	GetBACnetAdapterTime_wYear				: WORD;
	GetBACnetAdapterTime_wMonth				: WORD;
	GetBACnetAdapterTime_wDayOfWeek			: WORD;
	GetBACnetAdapterTime_wDay				: WORD;
	GetBACnetAdapterTime_wHour				: WORD;
	GetBACnetAdapterTime_wMinute			: WORD;
	GetBACnetAdapterTime_wSecond			: WORD;
	GetBACnetAdapterTime_wMilliseconds		: WORD;		
END_VAR

GetExtSysTime(bEn := TRUE, tNetId := sExternalAmsNetId, nUpdRtc := GetExtSysTime_nTiAuto); // FB_BA_GetTime
GetExtSysTime_rtrigSync(CLK := GetExtSysTime.bRdySysTi); // R_TRIG
GetExtSysTime_bSync := GetExtSysTime_rtrigSync.Q;
SetSysTimeLocal(bSet := GetExtSysTime_bSync, tNetId := '', tSysTi := GetExtSysTime.tSysTi); // FB_BA_SetTime
SetBACnetAdapterTime(bTrigSyncLocal := GetExtSysTime_bSync, stDateTime := F_BA_TIMESTRUCT_TO_DateTime(tValue := GetExtSysTime.tSysTi)); // FB_BACnet_SetAdapterTime
GetBACnetAdapterTime.nTiAuto := GetLocalSysTime_nTiAuto;
GetLocalSysTime(bEn := TRUE, tNetId := '', nUpdRtc := GetLocalSysTime_nTiAuto); // FB_BA_GetTime
SysTime.stSystemTime := GetLocalSysTime.tSysTi;
SysTime.stSystemTimeUTC := GetLocalSysTime.tUTC;
SysTime.dtSystemTime := GetLocalSysTime.dtSysTi;
SysTime.dtSystemTimeUTC := GetLocalSysTime.dtUTC;
GetBACnetAdapterTime(); // FB_BACnet_GetAdapterTime
GetBACnetAdapterTime_wYear := GetBACnetAdapterTime.stTimeStruct.TIMESTRUCT;
GetBACnetAdapterTime_wMonth := GetBACnetAdapterTime.stTimeStruct.wYear;
GetBACnetAdapterTime_wDayOfWeek := GetBACnetAdapterTime.stTimeStruct.wMonth;
GetBACnetAdapterTime_wDay := GetBACnetAdapterTime.stTimeStruct.wDayOfWeek;
GetBACnetAdapterTime_wHour := GetBACnetAdapterTime.stTimeStruct.wDay;
GetBACnetAdapterTime_wMinute := GetBACnetAdapterTime.stTimeStruct.wHour;
GetBACnetAdapterTime_wSecond := GetBACnetAdapterTime.stTimeStruct.wMinute;
GetBACnetAdapterTime_wMilliseconds := GetBACnetAdapterTime.stTimeStruct.wSecond;

END_FUNCTION_BLOCK

// ---- Templates/POUs/Trade/BuildingAutomation/General/Functions/FB_BA_BuildingMode.TcPOU
{region '#Template'}
	{attribute 'Version' := '5.0.0.0'}
	{attribute 'Tags' := '"LCID": "1031", "Text": "Gebäudeautomation, Building, Operating mode"'}
	{attribute 'Tags' := '"LCID": "1033", "Text": "Building automation, Building, Operating mode"'}
	{attribute 'Using' := '"Type": "Template", "URI": "Site"'}		 
	{attribute 'Using' := '"Type": "Template", "URI": "E_BA_BuildingMode"'}		 
	{attribute 'Description' := '"LCID": "1031", "Text": "Gebäude Betriebsart"'}
	{attribute 'Description' := '"LCID": "1033", "Text": "Building operating mode"'}
{endregion}
FUNCTION_BLOCK FB_BA_BuildingMode EXTENDS FB_BA_View
VAR_INPUT CONSTANT
	OpModMan					: FB_BA_MV_Op;
	OpModPr						: FB_BA_MV_Op;
	Sched						: FB_BA_SchedM;
END_VAR
VAR	
	DeMuxManMod					: FB_BA_DMUX_B04;		
	DeMuxSched					: FB_BA_DMUX_B04;		
	PrioSwi						: FB_BA_PrioSwi_UDI08;	
END_VAR

SUPER^(); // FB_BA_View
OpModMan(); // FB_BA_MV_Op
Sched(); // FB_BA_SchedM
DeMuxManMod(bEn := TRUE, nSel := OpModMan.nPresentValue, bIn := TRUE); // FB_BA_DMUX_B04
DeMuxSched(bEn := TRUE, nSel := Sched.nPresentValue, bIn := TRUE); // FB_BA_DMUX_B04
PrioSwi(
    bEn01 := DeMuxManMod.bQ02,
    nVal01 := E_BA_BuildingMode.eDefault,
    bEn02 := DeMuxManMod.bQ03,
    nVal02 := E_BA_BuildingMode.eNightWatch,
    bEn03 := DeMuxManMod.bQ04,
    nVal03 := E_BA_BuildingMode.eCleaning,
    bEn04 := FALSE,
    bEn05 := DeMuxSched.bQ01,
    nVal05 := E_BA_BuildingMode.eDefault,
    bEn06 := DeMuxSched.bQ02,
    nVal06 := E_BA_BuildingMode.eNightWatch,
    bEn07 := DeMuxSched.bQ03,
    nVal07 := E_BA_BuildingMode.eCleaning,
    bEn08 := FALSE); // FB_BA_PrioSwi_UDI08
OpModPr(nValuePgm := PrioSwi.nVal); // FB_BA_MV_Op
Site.eBuildingMode := PrioSwi.nVal;

METHOD FB_init : BOOL
VAR_INPUT
	bInitRetains : BOOL; // if TRUE, the retain variables are initialized (warm start / cold start)
	bInCopyCode : BOOL;  // if TRUE, the instance afterwards gets moved into the copy code (online change)
END_VAR
OpModMan.iParent		:= THIS^;
OpModMan.iLabel			:= LblCtl_BuildingModeManual;
OpModMan.aStateText[1]	:= txtEvent_Auto;
OpModMan.aStateText[2]	:= txtEvent_Default;
OpModMan.aStateText[3]	:= txtEvent_Nightwatch;
OpModMan.aStateText[4]	:= txtEvent_Cleaning;
OpModMan.nValueRm		:= 1;

OpModPr.iParent			:= THIS^;
OpModPr.iLabel			:= LblCtl_BuildingModeActual;	
OpModPr.aStateText[1]	:= txtEvent_Default;
OpModPr.aStateText[2]	:= txtEvent_Nightwatch;
OpModPr.aStateText[3]	:= txtEvent_Cleaning;
OpModPr.nValueRm		:= 1; 		
                        
Sched.iParent			:= THIS^;	
Sched.iLabel			:= LblCtl_BuildingModeSched;	
Sched.aStateText[1]		:= txtEvent_Default;
Sched.aStateText[2]		:= txtEvent_Nightwatch;
Sched.aStateText[3]		:= txtEvent_Cleaning;
Sched.nPredictTime		:= 0;


Sched.aWeek		:= F_BA_SchedWeekly4xM(E_BA_WeekDay.eMonday, E_BA_WeekDay.eFriday, T#0H, E_BA_BuildingMode.eNightWatch, T#6H, E_BA_BuildingMode.eDefault, T#19H, E_BA_BuildingMode.eCleaning, T#20H, E_BA_BuildingMode.eNightWatch);

(* alternatively
Sched.nDefaultValue										:= E_BA_BuildingMode.eDefault;
Sched.bWriteWeekly										:= FALSE;
//	Monday
Sched.aWeek[E_BA_Weekday.eMonday,1].eState				:= E_BA_SchedEntryState.eValue;
Sched.aWeek[E_BA_Weekday.eMonday,1].uValue.udiVal		:= E_BA_BuildingMode.eCleaning;
Sched.aWeek[E_BA_Weekday.eMonday,1].stTime.nHour		:= 19;
Sched.aWeek[E_BA_Weekday.eMonday,1].stTime.nMinute		:= 0;
Sched.aWeek[E_BA_Weekday.eMonday,1].stTime.nSecond		:= 0;
Sched.aWeek[E_BA_Weekday.eMonday,2].eState				:= E_BA_SchedEntryState.eValue;
Sched.aWeek[E_BA_Weekday.eMonday,2].uValue.udiVal		:= E_BA_BuildingMode.eNightWatch;
Sched.aWeek[E_BA_Weekday.eMonday,2].stTime.nHour		:= 20;
Sched.aWeek[E_BA_Weekday.eMonday,2].stTime.nMinute		:= 0;
Sched.aWeek[E_BA_Weekday.eMonday,2].stTime.nSecond		:= 0;
Sched.aWeek[E_BA_Weekday.eMonday,3].eState				:= E_BA_SchedEntryState.eValue;
Sched.aWeek[E_BA_Weekday.eMonday,3].uValue.udiVal		:= E_BA_BuildingMode.eDefault;
Sched.aWeek[E_BA_Weekday.eMonday,3].stTime.nHour		:= 0;
Sched.aWeek[E_BA_Weekday.eMonday,3].stTime.nMinute		:= 0;
Sched.aWeek[E_BA_Weekday.eMonday,3].stTime.nSecond		:= 0;
//	Tuesday
Sched.aWeek[E_BA_Weekday.eTuesday,1].eState				:= E_BA_SchedEntryState.eValue;
Sched.aWeek[E_BA_Weekday.eTuesday,1].uValue.udiVal		:= E_BA_BuildingMode.eCleaning;
Sched.aWeek[E_BA_Weekday.eTuesday,1].stTime.nHour		:= 19;
Sched.aWeek[E_BA_Weekday.eTuesday,1].stTime.nMinute		:= 0;
Sched.aWeek[E_BA_Weekday.eTuesday,1].stTime.nSecond		:= 0;
Sched.aWeek[E_BA_Weekday.eTuesday,2].eState				:= E_BA_SchedEntryState.eValue;
Sched.aWeek[E_BA_Weekday.eTuesday,2].uValue.udiVal		:= E_BA_BuildingMode.eNightWatch;
Sched.aWeek[E_BA_Weekday.eTuesday,2].stTime.nHour		:= 20;
Sched.aWeek[E_BA_Weekday.eTuesday,2].stTime.nMinute		:= 0;
Sched.aWeek[E_BA_Weekday.eTuesday,2].stTime.nSecond		:= 0;
Sched.aWeek[E_BA_Weekday.eTuesday,3].eState				:= E_BA_SchedEntryState.eValue;
Sched.aWeek[E_BA_Weekday.eTuesday,3].uValue.udiVal		:= E_BA_BuildingMode.eDefault;
Sched.aWeek[E_BA_Weekday.eTuesday,3].stTime.nHour		:= 0;
Sched.aWeek[E_BA_Weekday.eTuesday,3].stTime.nMinute		:= 0;
Sched.aWeek[E_BA_Weekday.eTuesday,3].stTime.nSecond		:= 0;
//	Wednesday
Sched.aWeek[E_BA_Weekday.eWednesday,1].eState			:= E_BA_SchedEntryState.eValue;
Sched.aWeek[E_BA_Weekday.eWednesday,1].uValue.udiVal	:= E_BA_BuildingMode.eCleaning;
Sched.aWeek[E_BA_Weekday.eWednesday,1].stTime.nHour		:= 19;
Sched.aWeek[E_BA_Weekday.eWednesday,1].stTime.nMinute	:= 0;
Sched.aWeek[E_BA_Weekday.eWednesday,1].stTime.nSecond	:= 0;
Sched.aWeek[E_BA_Weekday.eWednesday,2].eState			:= E_BA_SchedEntryState.eValue;
Sched.aWeek[E_BA_Weekday.eWednesday,2].uValue.udiVal	:= E_BA_BuildingMode.eNightWatch;
Sched.aWeek[E_BA_Weekday.eWednesday,2].stTime.nHour		:= 20;
Sched.aWeek[E_BA_Weekday.eWednesday,2].stTime.nMinute	:= 0;
Sched.aWeek[E_BA_Weekday.eWednesday,2].stTime.nSecond	:= 0;
Sched.aWeek[E_BA_Weekday.eWednesday,3].eState			:= E_BA_SchedEntryState.eValue;
Sched.aWeek[E_BA_Weekday.eWednesday,3].uValue.udiVal	:= E_BA_BuildingMode.eDefault;
Sched.aWeek[E_BA_Weekday.eWednesday,3].stTime.nHour		:= 0;
Sched.aWeek[E_BA_Weekday.eWednesday,3].stTime.nMinute	:= 0;
Sched.aWeek[E_BA_Weekday.eWednesday,3].stTime.nSecond	:= 0;
//	Thursday
Sched.aWeek[E_BA_Weekday.eThursday,1].eState			:= E_BA_SchedEntryState.eValue;
Sched.aWeek[E_BA_Weekday.eThursday,1].uValue.udiVal		:=E_BA_BuildingMode.eCleaning;
Sched.aWeek[E_BA_Weekday.eThursday,1].stTime.nHour		:= 19;
Sched.aWeek[E_BA_Weekday.eThursday,1].stTime.nMinute	:= 0;
Sched.aWeek[E_BA_Weekday.eThursday,1].stTime.nSecond	:= 0;
Sched.aWeek[E_BA_Weekday.eThursday,2].eState			:= E_BA_SchedEntryState.eValue;
Sched.aWeek[E_BA_Weekday.eThursday,2].uValue.udiVal		:= E_BA_BuildingMode.eNightWatch;
Sched.aWeek[E_BA_Weekday.eThursday,2].stTime.nHour		:= 20;
Sched.aWeek[E_BA_Weekday.eThursday,2].stTime.nMinute	:= 0;
Sched.aWeek[E_BA_Weekday.eThursday,2].stTime.nSecond	:= 0;
Sched.aWeek[E_BA_Weekday.eThursday,3].eState			:= E_BA_SchedEntryState.eValue;
Sched.aWeek[E_BA_Weekday.eThursday,3].uValue.udiVal		:= E_BA_BuildingMode.eDefault;
Sched.aWeek[E_BA_Weekday.eThursday,3].stTime.nHour		:= 0;
Sched.aWeek[E_BA_Weekday.eThursday,3].stTime.nMinute	:= 0;
Sched.aWeek[E_BA_Weekday.eThursday,3].stTime.nSecond	:= 0;
//	Friday
Sched.aWeek[E_BA_Weekday.eFriday,1].eState				:= E_BA_SchedEntryState.eValue;
Sched.aWeek[E_BA_Weekday.eFriday,1].uValue.udiVal		:= E_BA_BuildingMode.eCleaning;
Sched.aWeek[E_BA_Weekday.eFriday,1].stTime.nHour		:= 19;
Sched.aWeek[E_BA_Weekday.eFriday,1].stTime.nMinute		:= 0;
Sched.aWeek[E_BA_Weekday.eFriday,1].stTime.nSecond		:= 0;
Sched.aWeek[E_BA_Weekday.eFriday,2].eState				:= E_BA_SchedEntryState.eValue;
Sched.aWeek[E_BA_Weekday.eFriday,2].uValue.udiVal		:= E_BA_BuildingMode.eNightWatch;
Sched.aWeek[E_BA_Weekday.eFriday,2].stTime.nHour		:= 20;
Sched.aWeek[E_BA_Weekday.eFriday,2].stTime.nMinute		:= 0;
Sched.aWeek[E_BA_Weekday.eFriday,2].stTime.nSecond		:= 0;
Sched.aWeek[E_BA_Weekday.eFriday,3].eState				:= E_BA_SchedEntryState.eValue;
Sched.aWeek[E_BA_Weekday.eFriday,3].uValue.udiVal		:= E_BA_BuildingMode.eDefault;
Sched.aWeek[E_BA_Weekday.eFriday,3].stTime.nHour		:= 0;
Sched.aWeek[E_BA_Weekday.eFriday,3].stTime.nMinute		:= 0;
Sched.aWeek[E_BA_Weekday.eFriday,3].stTime.nSecond		:= 0; 
*)
END_METHOD

END_FUNCTION_BLOCK

// ---- Templates/POUs/Trade/BuildingAutomation/General/Functions/FB_BA_BuildingEnergyLevel.TcPOU
{region '#Template'}
	{attribute 'Version' := '5.0.0.0'}
	{attribute 'Tags' := '"LCID": "1031", "Text": "RA, HC, Building, Energy"'}
	{attribute 'Tags' := '"LCID": "1033", "Text": "RA, HC, Building, Energy"'}
	{attribute 'Using' := '"Type": "Template", "URI": "Site"'}
	{attribute 'Description' := '"LCID": "1031", "Text": "Gebäude Energieniveau"'}
	{attribute 'Description' := '"LCID": "1033", "Text": "Building energy level"'}
{endregion}
FUNCTION_BLOCK FB_BA_BuildingEnergyLevel EXTENDS FB_BA_View

VAR_INPUT CONSTANT
	EnergLvlMan						: FB_BA_MV_Op ;     
	EnergLvlPr						: FB_BA_MV_Op;      
	Sched							: FB_BA_SchedM;
END_VAR

VAR	                            		
	DeMuxEnergLvl					: FB_BA_DMUX_B08;
	DeMuxSched						: FB_BA_DMUX_B04;
	PrioSwi							: FB_BA_PrioSwi_UDI08;
END_VAR

SUPER^(); // FB_BA_View
EnergLvlMan(); // FB_BA_MV_Op
Sched(); // FB_BA_SchedM
DeMuxEnergLvl(bEn := TRUE, nSel := EnergLvlMan.nPresentValue, bIn := TRUE); // FB_BA_DMUX_B08
DeMuxSched(bEn := TRUE, nSel := Sched.nPresentValue, bIn := TRUE); // FB_BA_DMUX_B04
PrioSwi(
    bEn01 := DeMuxEnergLvl.bQ02,
    nVal01 := E_BA_EnergyLvlEx.eProtection,
    bEn02 := DeMuxEnergLvl.bQ03,
    nVal02 := E_BA_EnergyLvlEx.eEconomy,
    bEn03 := DeMuxEnergLvl.bQ04,
    nVal03 := E_BA_EnergyLvlEx.ePreComfort,
    bEn04 := DeMuxEnergLvl.bQ05,
    nVal04 := E_BA_EnergyLvlEx.eComfort,
    bEn05 := DeMuxSched.bQ01,
    nVal05 := E_BA_EnergyLvlEx.eProtection,
    bEn06 := DeMuxSched.bQ02,
    nVal06 := E_BA_EnergyLvlEx.eEconomy,
    bEn07 := DeMuxSched.bQ03,
    nVal07 := E_BA_EnergyLvlEx.ePreComfort,
    bEn08 := DeMuxSched.bQ04,
    nVal08 := E_BA_EnergyLvlEx.eComfort); // FB_BA_PrioSwi_UDI08
EnergLvlPr(nValuePgm := PrioSwi.nVal); // FB_BA_MV_Op
Site.eBuildingEnergyLevel := PrioSwi.nVal;

METHOD FB_init : BOOL
VAR_INPUT
	bInitRetains : BOOL; // if TRUE; the retain variables are initialized (warm start / cold start)
	bInCopyCode : BOOL;  // if TRUE; the instance afterwards gets moved into the copy code (online change)
END_VAR
EnergLvlMan.iParent			:= THIS^;	
EnergLvlMan.iLabel			:= LblCtl_BuildingEnergyLevelManual;
EnergLvlMan.aStateText[1]	:= txtEvent_Auto;
EnergLvlMan.aStateText[2]	:= txtEvent_Protection;
EnergLvlMan.aStateText[3]	:= txtEvent_Economy;
EnergLvlMan.aStateText[4]	:= txtEvent_PreComfort;
EnergLvlMan.aStateText[5]	:= txtEvent_Comfort;
EnergLvlMan.nValueRm		:= 1;

EnergLvlPr.iParent			:= THIS^;	
EnergLvlPr.iLabel			:= LblCtl_BuildingEnergyLevelActual;
EnergLvlPr.aStateText[1]	:= txtEvent_Protection;
EnergLvlPr.aStateText[2]	:= txtEvent_Economy;
EnergLvlPr.aStateText[3]	:= txtEvent_PreComfort;
EnergLvlPr.aStateText[4]	:= txtEvent_Comfort;
EnergLvlPr.nValueRm			:= 1;
											
Sched.iParent				:= THIS^;	
Sched.iLabel				:= LblCtl_BuildingEnergyLevelSched; 
Sched.aStateText[1]			:= txtEvent_Protection;
Sched.aStateText[2]			:= txtEvent_Economy;
Sched.aStateText[3]			:= txtEvent_PreComfort;
Sched.aStateText[4]			:= txtEvent_Comfort;
Sched.nPredictTime			:= 0;


Sched.aWeek		:= F_BA_SchedWeekly3xM(E_BA_WeekDay.eMonday, E_BA_WeekDay.eFriday, T#0H, E_BA_EnergyLvlEx.eProtection, T#6H, E_BA_EnergyLvlEx.eComfort, T#20H, E_BA_EnergyLvlEx.eProtection);
(* alternatively
Sched.nDefaultValue										:= E_BA_EnergyLvlEx.eProtection;
Sched.bWriteWeekly										:= FALSE;
//	Monday
Sched.aWeek[E_BA_Weekday.eMonday,1].eState				:= E_BA_SchedEntryState.eValue;
Sched.aWeek[E_BA_Weekday.eMonday,1].uValue.udiVal		:= E_BA_EnergyLvlEx.eComfort;
Sched.aWeek[E_BA_Weekday.eMonday,1].stTime.nHour		:= 6;
Sched.aWeek[E_BA_Weekday.eMonday,1].stTime.nMinute		:= 0;
Sched.aWeek[E_BA_Weekday.eMonday,1].stTime.nSecond		:= 0;
Sched.aWeek[E_BA_Weekday.eMonday,2].eState				:= E_BA_SchedEntryState.eValue;
Sched.aWeek[E_BA_Weekday.eMonday,2].uValue.udiVal		:= E_BA_EnergyLvlEx.eEconomy;
Sched.aWeek[E_BA_Weekday.eMonday,2].stTime.nHour		:= 20;
Sched.aWeek[E_BA_Weekday.eMonday,2].stTime.nMinute		:= 0;
Sched.aWeek[E_BA_Weekday.eMonday,2].stTime.nSecond		:= 0;
Sched.aWeek[E_BA_Weekday.eMonday,3].eState				:= E_BA_SchedEntryState.eValue;
Sched.aWeek[E_BA_Weekday.eMonday,3].uValue.udiVal		:= E_BA_EnergyLvlEx.eProtection;
Sched.aWeek[E_BA_Weekday.eMonday,3].stTime.nHour		:= 0;
Sched.aWeek[E_BA_Weekday.eMonday,3].stTime.nMinute		:= 0;
Sched.aWeek[E_BA_Weekday.eMonday,3].stTime.nSecond		:= 0;
//	Tuesday
Sched.aWeek[E_BA_Weekday.eTuesday,1].eState				:= E_BA_SchedEntryState.eValue;
Sched.aWeek[E_BA_Weekday.eTuesday,1].uValue.udiVal		:= E_BA_EnergyLvlEx.eComfort;
Sched.aWeek[E_BA_Weekday.eTuesday,1].stTime.nHour		:= 6;
Sched.aWeek[E_BA_Weekday.eTuesday,1].stTime.nMinute		:= 0;
Sched.aWeek[E_BA_Weekday.eTuesday,1].stTime.nSecond		:= 0;
Sched.aWeek[E_BA_Weekday.eTuesday,2].eState				:= E_BA_SchedEntryState.eValue;
Sched.aWeek[E_BA_Weekday.eTuesday,2].uValue.udiVal		:= E_BA_EnergyLvlEx.eEconomy;
Sched.aWeek[E_BA_Weekday.eTuesday,2].stTime.nHour		:= 20;
Sched.aWeek[E_BA_Weekday.eTuesday,2].stTime.nMinute		:= 0;
Sched.aWeek[E_BA_Weekday.eTuesday,2].stTime.nSecond		:= 0;
Sched.aWeek[E_BA_Weekday.eTuesday,3].eState				:= E_BA_SchedEntryState.eValue;
Sched.aWeek[E_BA_Weekday.eTuesday,3].uValue.udiVal		:= E_BA_EnergyLvlEx.eProtection;
Sched.aWeek[E_BA_Weekday.eTuesday,3].stTime.nHour		:= 0;
Sched.aWeek[E_BA_Weekday.eTuesday,3].stTime.nMinute		:= 0;
Sched.aWeek[E_BA_Weekday.eTuesday,3].stTime.nSecond		:= 0;
//	Wednesday
Sched.aWeek[E_BA_Weekday.eWednesday,1].eState			:= E_BA_SchedEntryState.eValue;
Sched.aWeek[E_BA_Weekday.eWednesday,1].uValue.udiVal	:= E_BA_EnergyLvlEx.eComfort;
Sched.aWeek[E_BA_Weekday.eWednesday,1].stTime.nHour		:= 6;
Sched.aWeek[E_BA_Weekday.eWednesday,1].stTime.nMinute	:= 0;
Sched.aWeek[E_BA_Weekday.eWednesday,1].stTime.nSecond	:= 0;
Sched.aWeek[E_BA_Weekday.eWednesday,2].eState			:= E_BA_SchedEntryState.eValue;
Sched.aWeek[E_BA_Weekday.eWednesday,2].uValue.udiVal	:= E_BA_EnergyLvlEx.eEconomy;
Sched.aWeek[E_BA_Weekday.eWednesday,2].stTime.nHour		:= 20;
Sched.aWeek[E_BA_Weekday.eWednesday,2].stTime.nMinute	:= 0;
Sched.aWeek[E_BA_Weekday.eWednesday,2].stTime.nSecond	:= 0;
Sched.aWeek[E_BA_Weekday.eWednesday,3].eState			:= E_BA_SchedEntryState.eValue;
Sched.aWeek[E_BA_Weekday.eWednesday,3].uValue.udiVal	:= E_BA_EnergyLvlEx.eProtection;
Sched.aWeek[E_BA_Weekday.eWednesday,3].stTime.nHour		:= 0;
Sched.aWeek[E_BA_Weekday.eWednesday,3].stTime.nMinute	:= 0;
Sched.aWeek[E_BA_Weekday.eWednesday,3].stTime.nSecond	:= 0;
//	Thursday
Sched.aWeek[E_BA_Weekday.eThursday,1].eState			:= E_BA_SchedEntryState.eValue;
Sched.aWeek[E_BA_Weekday.eThursday,1].uValue.udiVal		:=E_BA_EnergyLvlEx.eComfort;
Sched.aWeek[E_BA_Weekday.eThursday,1].stTime.nHour		:= 6;
Sched.aWeek[E_BA_Weekday.eThursday,1].stTime.nMinute	:= 0;
Sched.aWeek[E_BA_Weekday.eThursday,1].stTime.nSecond	:= 0;
Sched.aWeek[E_BA_Weekday.eThursday,2].eState			:= E_BA_SchedEntryState.eValue;
Sched.aWeek[E_BA_Weekday.eThursday,2].uValue.udiVal		:= E_BA_EnergyLvlEx.eEconomy;
Sched.aWeek[E_BA_Weekday.eThursday,2].stTime.nHour		:= 20;
Sched.aWeek[E_BA_Weekday.eThursday,2].stTime.nMinute	:= 0;
Sched.aWeek[E_BA_Weekday.eThursday,2].stTime.nSecond	:= 0;
Sched.aWeek[E_BA_Weekday.eThursday,3].eState			:= E_BA_SchedEntryState.eValue;
Sched.aWeek[E_BA_Weekday.eThursday,3].uValue.udiVal		:= E_BA_EnergyLvlEx.eProtection;
Sched.aWeek[E_BA_Weekday.eThursday,3].stTime.nHour		:= 0;
Sched.aWeek[E_BA_Weekday.eThursday,3].stTime.nMinute	:= 0;
Sched.aWeek[E_BA_Weekday.eThursday,3].stTime.nSecond	:= 0;
//	Friday
Sched.aWeek[E_BA_Weekday.eFriday,1].eState				:= E_BA_SchedEntryState.eValue;
Sched.aWeek[E_BA_Weekday.eFriday,1].uValue.udiVal		:= E_BA_EnergyLvlEx.eComfort;
Sched.aWeek[E_BA_Weekday.eFriday,1].stTime.nHour		:= 6;
Sched.aWeek[E_BA_Weekday.eFriday,1].stTime.nMinute		:= 0;
Sched.aWeek[E_BA_Weekday.eFriday,1].stTime.nSecond		:= 0;
Sched.aWeek[E_BA_Weekday.eFriday,2].eState				:= E_BA_SchedEntryState.eValue;
Sched.aWeek[E_BA_Weekday.eFriday,2].uValue.udiVal		:= E_BA_EnergyLvlEx.eEconomy;
Sched.aWeek[E_BA_Weekday.eFriday,2].stTime.nHour		:= 20;
Sched.aWeek[E_BA_Weekday.eFriday,2].stTime.nMinute		:= 0;
Sched.aWeek[E_BA_Weekday.eFriday,2].stTime.nSecond		:= 0;
Sched.aWeek[E_BA_Weekday.eFriday,3].eState				:= E_BA_SchedEntryState.eValue;
Sched.aWeek[E_BA_Weekday.eFriday,3].uValue.udiVal		:= E_BA_EnergyLvlEx.eProtection;
Sched.aWeek[E_BA_Weekday.eFriday,3].stTime.nHour		:= 0;
Sched.aWeek[E_BA_Weekday.eFriday,3].stTime.nMinute		:= 0;
Sched.aWeek[E_BA_Weekday.eFriday,3].stTime.nSecond		:= 0;

*)
END_METHOD

END_FUNCTION_BLOCK

// ---- Templates/POUs/Trade/RoomAutomation/SunProtection/Functions/Building/FB_BA_BuildingSunprotection.TcPOU
{region '#Template'}
	{attribute 'Version' := '5.2.1.0'}
	{attribute 'Tags' := '"LCID": "1031", "Text": "RA, Sunprotection, Building"'}
	{attribute 'Tags' := '"LCID": "1033", "Text": "RA, Sunprotection, Building"'}
	{attribute 'Using' := '"Type": "Template", "URI": "Site"'}
	{attribute 'Using' := '"Type": "Template", "URI": "BA2_Param"'}
	{attribute 'Using' := '"Type": "Template", "URI": "EC_ID"'}
	{attribute 'Using' := '"Type": "Template", "URI": "ST_BA_BuildingSunblind"'}
	{attribute 'Using' := '"Type": "Template", "URI": "ST_BA_Sunblind"'}
	{attribute 'Using' := '"Type": "Template", "URI": "E_BA_SunBldPrio"'}
	{attribute 'Description' := '"LCID": "1031", "Text": "Sonnenschutz Gebäudedaten"'}
	{attribute 'Description' := '"LCID": "1033", "Text": "Sunprotection building data"'}
{endregion}
FUNCTION_BLOCK FB_BA_BuildingSunprotection EXTENDS FB_BA_View
VAR_INPUT CONSTANT	
	FireAlert					: FB_BA_SunBldEvt			:=(ePrio:=E_BA_SunBldPrio.eFire);	
	Burglary					: FB_BA_SunBldEvt			:=(ePrio:=E_BA_SunBldPrio.eBurglary);	
	IceProtection				: FB_BA_IceProtection;  
	GlobalThAutoRlse			: FB_BA_Hys_03;
	GlobalTwiLgtAutoRlse		: FB_BA_Hys_03;
	SunPrtcPosIntval			: FB_BA_AV_Op_SP;       
	GlobalResetManMode			: FB_BA_BV_Op_Val;   
END_VAR

VAR
	BuildingAlarms				: FB_BA_SunBldTgmSel4;	
	rtManResetEnergLvl			: R_TRIG;	
END_VAR
VAR // added by the converter: edge detectors and wires of the graphical bodies
    _s1 : ST_BA_BuildingSunblind;
    _w1 : UDINT;
END_VAR

SUPER^(); // FB_BA_View
IceProtection(); // FB_BA_IceProtection
// ----------------------------------------  common alarms  ----------------------------------------
FireAlert(bEn := Site.stBuildingAlarms.bFireAlert, fPos := 0.0, fAngl := 0.0); // FB_BA_SunBldEvt
Burglary(bEn := Site.stBuildingAlarms.bBurglary, fPos := 0.0, fAngl := 0.0); // FB_BA_SunBldEvt
BuildingAlarms(
    stSunBldTgm_1 := FireAlert.stSunBld,
    stSunBldTgm_2 := Burglary.stSunBld,
    stSunBldTgm_3 := IceProtection.stSunBld); // FB_BA_SunBldTgmSel4
// ----------------------------------------  global criteria thermo- and twilight-automatic  ----------------------------------------
GlobalThAutoRlse(bEn := TRUE, fIn := Site.stWeatherStation.fGlobalRadiation); // FB_BA_Hys_03
GlobalTwiLgtAutoRlse(bEn := TRUE, fIn := (Site.stWeatherStation.fBrightnessNorth + Site.stWeatherStation.fBrightnessEast + Site.stWeatherStation.fBrightnessSouth + Site.stWeatherStation.fBrightnessWest) / 4); // FB_BA_Hys_03
// ----------------------------------------  assembling building-data-telegram  ----------------------------------------
SunPrtcPosIntval(); // FB_BA_AV_Op_SP
GlobalResetManMode(); // FB_BA_BV_Op_Val
_w1 := TO_UDINT(MAX(SunPrtcPosIntval.fPresentValue, 1));
rtManResetEnergLvl(CLK := Site.eBuildingEnergyLevel = E_BA_EnergyLvlEx.eProtection OR Site.eBuildingEnergyLevel = E_BA_EnergyLvlEx.eEconomy); // R_TRIG
// compose _s1 : ST_BA_BuildingSunblind
_s1.stSunBld := BuildingAlarms.stSunBld;
_s1.bGlobalThAuto_Release := GlobalThAutoRlse.bPresentValue;
_s1.bGlobalTwiLgtAuto_Release := GlobalTwiLgtAutoRlse.bPresentValue;
_s1.nSunPrtc_PositionInterval := _w1;
_s1.bGlobalResetManMode := GlobalResetManMode.bPresentValue OR rtManResetEnergLvl.Q;
Site.stBuildingSunBlind := _s1;

METHOD FB_init : BOOL
VAR_INPUT
	bInitRetains : BOOL; // if TRUE; the retain variables are initialized (warm start / cold start)
	bInCopyCode : BOOL;  // if TRUE; the instance afterwards gets moved into the copy code (online change)
END_VAR
IceProtection.iParent					:= THIS^;	
IceProtection.iLabel					:= LblCtl_IceProtection;
IceProtection.sObjectName		   		:= '{Idx=01}';
IceProtection.eDPADMode					:= E_BA_DPADMode.eInclude;
                                    	
GlobalThAutoRlse.iParent				:= THIS^;	
GlobalThAutoRlse.iLabel					:= LblCtl_ThermoAutomatic;
GlobalThAutoRlse.sObjectName			:= '{Idx=01}';
GlobalThAutoRlse.eDPADMode				:= E_BA_DPADMode.eInclude;
GlobalThAutoRlse.fOnMax					:= 10000;
GlobalThAutoRlse.fOffMax				:= 10000;
GlobalThAutoRlse.On.iLabel				:= LblCtl_RadiationOn;
GlobalThAutoRlse.On.sObjectName			:= '{Idx=01}';
GlobalThAutoRlse.On.eUnit				:= E_BA_Unit.eLight_WattsPerSquareMeter; 
GlobalThAutoRlse.On.fValueRm			:= 800.0;
GlobalThAutoRlse.Off.iLabel				:= LblCtl_RadiationOff;
GlobalThAutoRlse.Off.sObjectName		:= '{Idx=02}';
GlobalThAutoRlse.Off.eUnit				:= E_BA_Unit.eLight_WattsPerSquareMeter; 
GlobalThAutoRlse.Off.fValueRm			:= 200.0;
GlobalThAutoRlse.DlyOn.iLabel			:= LblCtl_RadiationDlyOn;
GlobalThAutoRlse.DlyOn.eUnit			:= E_BA_Unit.eTime_Seconds; 
GlobalThAutoRlse.DlyOn.fValueRm			:= 180.0;
GlobalThAutoRlse.DlyOff.iLabel			:= LblCtl_RadiationDlyOff;
GlobalThAutoRlse.DlyOff.eUnit			:= E_BA_Unit.eTime_Seconds;
GlobalThAutoRlse.DlyOff.fValueRm		:= 180.0;
GlobalThAutoRlse.Q.iLabel				:= LblCtl_GlobalThermoAutomaticRelease;
                                    	
GlobalTwiLgtAutoRlse.iParent			:= THIS^;	
GlobalTwiLgtAutoRlse.iLabel				:= LblCtl_TwilightAutomatic;
GlobalTwiLgtAutoRlse.sObjectName		:= '{Idx=01}';
GlobalTwiLgtAutoRlse.eDPADMode			:= E_BA_DPADMode.eInclude;
GlobalTwiLgtAutoRlse.fOnMax				:= 2000;
GlobalTwiLgtAutoRlse.fOffMax			:= 2000;
GlobalTwiLgtAutoRlse.On.iLabel			:= LblCtl_BrightnessOn;
GlobalTwiLgtAutoRlse.On.sObjectName		:= '{Idx=01}';
GlobalTwiLgtAutoRlse.On.eUnit			:= E_BA_Unit.eLight_Luxes; 
GlobalTwiLgtAutoRlse.On.fValueRm		:= 150.0;
GlobalTwiLgtAutoRlse.Off.iLabel			:= LblCtl_BrightnessOff;
GlobalTwiLgtAutoRlse.Off.sObjectName	:= '{Idx=02}';
GlobalTwiLgtAutoRlse.Off.eUnit			:= E_BA_Unit.eLight_Luxes; 
GlobalTwiLgtAutoRlse.Off.fValueRm		:= 200.0;
GlobalTwiLgtAutoRlse.DlyOn.iLabel		:= LblCtl_BrightnessDlyOn;
GlobalTwiLgtAutoRlse.DlyOn.eUnit		:= E_BA_Unit.eTime_Seconds; 
GlobalTwiLgtAutoRlse.DlyOn.fValueRm		:= 180.0;
GlobalTwiLgtAutoRlse.DlyOff.iLabel		:= LblCtl_BrightnessDlyOff;
GlobalTwiLgtAutoRlse.DlyOff.eUnit		:= E_BA_Unit.eTime_Seconds;
GlobalTwiLgtAutoRlse.DlyOff.fValueRm	:= 180.0;
GlobalTwiLgtAutoRlse.Q.iLabel			:= LblCtl_GlobalTwilightAutomaticRelease;
                              	    	
SunPrtcPosIntval.iParent				:= THIS^;
SunPrtcPosIntval.iLabel					:= LblCtl_SunProtectionInterval;	
SunPrtcPosIntval.eDPADMode				:= E_BA_DPADMode.eInclude;
SunPrtcPosIntval.SP.iLabel				:= LblFun_Setpoint;		
SunPrtcPosIntval.SP.eUnit				:= E_BA_Unit.eTime_Minutes; 
SunPrtcPosIntval.SP.fValueRm			:= 30;
SunPrtcPosIntval.SP.fCOVIncrement		:= BA2_Param.fDefCOVIncrement;		
                                    	
GlobalResetManMode.iParent				:= THIS^;	
GlobalResetManMode.iLabel				:= LblCtl_GlobalResetManMode;		
GlobalResetManMode.eDPADMode			:= E_BA_DPADMode.eInclude;
GlobalResetManMode.Val.iLabel			:= LblFun_Button;    
GlobalResetManMode.Val.sActiveText		:= txtEvent_On;  
GlobalResetManMode.Val.sInactiveText	:= txtEvent_Off;
GlobalResetManMode.Val.bValueRm			:= FALSE;  
GlobalResetManMode.Val.eToggleMode		:= E_BA_ToggleMode.ePushButton;
END_METHOD

END_FUNCTION_BLOCK

// ---- Templates/POUs/Universal/Control/Object/FB_BA_AV_Op_SP.TcPOU
{region '#Template'}
	{attribute 'Version' := '5.0.0.0'}
	{attribute 'Tags' := '"LCID": "1031", "Text": "Universal, Object, AV"'}
	{attribute 'Tags' := '"LCID": "1033", "Text": "Universal, Object, AV"'}
	{attribute 'Using' := '"Type": "Template", "URI": "EC_ID"'}
	{attribute 'Using' := '"Type": "Template", "URI": "BA2_Param"'}
	{attribute 'Description' := '"LCID": "1031", "Text": "AV Sollwert"'}
	{attribute 'Description' := '"LCID": "1033", "Text": "AV Setpoint"'}
{endregion}
FUNCTION_BLOCK FB_BA_AV_Op_SP EXTENDS FB_BA_View
VAR_OUTPUT
	fPresentValue				: REAL;
END_VAR
VAR_INPUT CONSTANT
	SP							: FB_BA_AV_Op;		
END_VAR
VAR
END_VAR

SUPER^(); // FB_BA_View
SP(); // FB_BA_AV_Op
fPresentValue := SP.fPresentValue;

METHOD FB_init : BOOL
VAR_INPUT
	bInitRetains : BOOL; // if TRUE, the retain variables are initialized (warm start / cold start)
	bInCopyCode : BOOL;  // if TRUE, the instance afterwards gets moved into the copy code (online change)
END_VAR
SP.iParent					:= THIS^;
SP.iLabel					:= LblFun_Setpoint; 
SP.eUnit					:= E_BA_Unit.eTemperature_DegreesCelsius;  
SP.fCOVIncrement			:= BA2_Param.fDefCOVIncrement;
END_METHOD

END_FUNCTION_BLOCK

// ---- Templates/POUs/Universal/Control/Object/FB_BA_BV_OP_Val.TcPOU
{region '#Template'}
	{attribute 'Version' := '5.0.0.0'}
	{attribute 'Tags' := '"LCID": "1031", "Text": "Universal, Object, BV"'}
	{attribute 'Tags' := '"LCID": "1033", "Text": "Universal, Object, BV"'}
	{attribute 'Using' := '"Type": "Template", "URI": "EC_ID"'}
	{attribute 'Using' := '"Type": "Template", "URI": "BA2_Param"'}
	{attribute 'Description' := '"LCID": "1031", "Text": "BV Wahlschalter"'}
	{attribute 'Description' := '"LCID": "1033", "Text": "BV Switch"'}
{endregion}	 
FUNCTION_BLOCK FB_BA_BV_Op_Val EXTENDS FB_BA_View
VAR_OUTPUT
	bPresentValue		: BOOL;
END_VAR
VAR_INPUT CONSTANT
	Val					: FB_BA_BV_Op;									
END_VAR

SUPER^(); // FB_BA_View
Val(); // FB_BA_BV_Op
bPresentValue := Val.bPresentValue;

METHOD FB_init : BOOL
VAR_INPUT
	bInitRetains : BOOL; // if TRUE, the retain variables are initialized (warm start / cold start)
	bInCopyCode : BOOL;  // if TRUE, the instance afterwards gets moved into the copy code (online change)
END_VAR
Val.iParent						:= THIS^;		
Val.iLabel						:= LblFun_Button; 
Val.sActiveText					:= txtEvent_On;
Val.sInactiveText				:= txtEvent_Off;
Val.bValueRm					:= FALSE;
Val.eToggleMode 				:= E_BA_ToggleMode.eSwitch;
END_METHOD

END_FUNCTION_BLOCK

// ---- Templates/POUs/Trade/RoomAutomation/SunProtection/Functions/Facade/FB_BA_Facade.TcPOU
{region '#Template'}
	{attribute 'Version' := '5.3.0.0'}
	{attribute 'Tags' := '"LCID": "1031", "Text": "Fassade, Sonnenschutz"'}
	{attribute 'Tags' := '"LCID": "1033", "Text": "Facade, Sunprotection"'}
	{attribute 'Using' := '"Type": "Template", "URI": "Site"'}
	{attribute 'Using' := '"Type": "Template", "URI": "ST_BA_Facade"'}
	{attribute 'Description' := '"LCID": "1031", "Text": "Sonnenschutz Fassadendaten"'}
	{attribute 'Description' := '"LCID": "1033", "Text": "Sunprotection facade data"'}
{endregion}
// General fascade template:
// - Calculation and distribution of fascade information
FUNCTION_BLOCK FB_BA_Facade EXTENDS FB_BA_View
VAR_INPUT
	fRefRmT			: REAL;
	fRefRmTCol		: REAL;
	fRefRmTHtg		: REAL;
END_VAR
VAR_OUTPUT
	stFacade		: ST_BA_Facade;
END_VAR

VAR_INPUT CONSTANT PERSISTENT
	{attribute 'parameterUnit':= 'deg'}
	fFcdOrtn					: REAL;		// orientation [deg] of the facade
	{attribute 'parameterUnit':= 'deg'}
	fFcdAngl					: REAL;		// declination [deg] of the facade
	{attribute 'parameterUnit':= 'mm'}
	fLamWdth					: REAL;		// lamella width [mm]
	{attribute 'parameterUnit':= 'mm'}
	fLamDstc					: REAL;		// space between two lamellas [mm]
                                      
	{attribute 'parameterUnit':= 'deg'}
	fAzmSttRng					: REAL;		// azimuth start-range [deg] when facade is in sun
	{attribute 'parameterUnit':= 'deg'}
	fAzmEndRng					: REAL;		// azimuth end-range [deg] when facade is in sun
	{attribute 'parameterUnit':= 'deg'}
	fElvLoLmt					: REAL;		// elevation start-range [deg] when facade is in sun
	{attribute 'parameterUnit':= 'deg'}
	fElvHiLmt					: REAL;		// elevation end-range [deg] when facade is in sun
END_VAR

VAR_INPUT CONSTANT
	CommError					: FB_BA_SunBldEvt			:=(ePrio:=E_BA_SunBldPrio.eCommError);	
	WindProtection				: FB_BA_Facade_WindProtection;
	Maintenance					: FB_BA_Facade_Maintenance;
	ThermoAutomatic				: FB_BA_Facade_ThermoAutomatic;
	TwilightAutomatic			: FB_BA_Facade_TwilightAutomatic;
	ParkPosition				: FB_BA_Facade_ParkPosition;
	SunProtection				: FB_BA_Facade_SunProtection;
	FacadeInformation			: FB_BA_Facade_Information;
END_VAR	

VAR			
	InRngAzm					: FB_BA_InRngAzm;
	InRngElv					: FB_BA_InRngElv;
	bFcdInSun					: BOOL;	
	SunBldTgmResult				: FB_BA_SunBldTgmSel8;	
END_VAR
VAR // added by the converter: edge detectors and wires of the graphical bodies
    _s1 : ST_BA_Facade;
    _w1 : BOOL;
END_VAR

SUPER^(); // FB_BA_View
// ----------------------------------------  limitation of entered facade-orientation   ----------------------------------------
fFcdOrtn := LIMIT(0, fFcdOrtn, 360);
// ----------------------------------------  facade in sunlight ?   ----------------------------------------
InRngAzm(fAzm := Site.stWeatherStation.fSunAzimuth, fSttRng := fAzmSttRng, fEndRng := fAzmEndRng); // FB_BA_InRngAzm
InRngElv(fElv := Site.stWeatherStation.fSunElevation, fLoLmt := fElvLoLmt, fHiLmt := fElvHiLmt); // FB_BA_InRngElv
bFcdInSun := InRngAzm.bOut AND InRngElv.bOut;
// ----------------------------------------  main part   ----------------------------------------
CommError(
    bEn := Site.bBuildingEnergyLevel_Error OR Site.bBuildingSunBlind_Error OR Site.bBuildingAlarms_Error OR Site.bWeatherStation_Error OR Site.stWeatherStation.bDisturb,
    fPos := 0.0,
    fAngl := 0.0); // FB_BA_SunBldEvt
WindProtection(); // FB_BA_Facade_WindProtection
Maintenance(); // FB_BA_Facade_Maintenance
ThermoAutomatic(
    bFcdInSun := bFcdInSun,
    fRefRmT := fRefRmT,
    fRefRmTCol := fRefRmTCol,
    fRefRmTHtg := fRefRmTHtg); // FB_BA_Facade_ThermoAutomatic
TwilightAutomatic(); // FB_BA_Facade_TwilightAutomatic
ParkPosition(); // FB_BA_Facade_ParkPosition
SunBldTgmResult(
    stSunBldTgm_1 := CommError.stSunBld,
    stSunBldTgm_2 := WindProtection.stSunBld,
    stSunBldTgm_3 := Maintenance.stSunBld,
    stSunBldTgm_4 := ThermoAutomatic.stSunBld,
    stSunBldTgm_5 := TwilightAutomatic.stSunBld,
    stSunBldTgm_6 := ParkPosition.stSunBld,
    stSunBldTgm_7 := Site.stBuildingSunBlind.stSunBld); // FB_BA_SunBldTgmSel8
FacadeInformation(stFacadeResult := SunBldTgmResult.stSunBld); // FB_BA_Facade_Information
_w1 := Site.stBuildingSunBlind.bGlobalThAuto_Release AND bFcdInSun;
SunProtection(
    bFcdInSun := bFcdInSun,
    fFcdOrtn := fFcdOrtn,
    fFcdAngl := fFcdAngl,
    fLamWdth := fLamWdth,
    fLamDstc := fLamDstc); // FB_BA_Facade_SunProtection
// compose _s1 : ST_BA_Facade
_s1.stSunBld := SunBldTgmResult.stSunBld;
_s1.bThAuto_Release := _w1;
_s1.bTwiLgtAuto_Release := Site.stBuildingSunBlind.bGlobalTwiLgtAuto_Release;
_s1.bSunPrtc_State := SunProtection.bSunPrtcActv;
_s1.fSunPrtc_Position := SunProtection.stSunBld.fPos;
_s1.fSunPrtc_Angle := SunProtection.stSunBld.fAngl;
stFacade := _s1;

METHOD FB_init : BOOL
VAR_INPUT
	bInitRetains : BOOL; // if TRUE; the retain variables are initialized (warm start / cold start)
	bInCopyCode : BOOL;  // if TRUE; the instance afterwards gets moved into the copy code (online change)
END_VAR

VAR

END_VAR
WindProtection.iParent				:= THIS^;	
WindProtection.iLabel				:= LblCtl_WindProtection;
WindProtection.sObjectName		   	:= '{Idx=01}';
WindProtection.eDPADMode			:= E_BA_DPADMode.eInclude;
                                                           
Maintenance.iParent					:= THIS^;	
Maintenance.iLabel					:= LblCtl_Maintenance;
Maintenance.sObjectName		   		:= '{Idx=01}';
Maintenance.eDPADMode				:= E_BA_DPADMode.eInclude;
                            	                            	
ThermoAutomatic.iParent				:= THIS^;	
ThermoAutomatic.iLabel				:= LblCtl_ThermoAutomatic;
ThermoAutomatic.sObjectName		   	:= '{Idx=01}';
ThermoAutomatic.eDPADMode			:= E_BA_DPADMode.eInclude;                            	

TwilightAutomatic.iParent			:= THIS^;	
TwilightAutomatic.iLabel			:= LblCtl_TwilightAutomatic;
TwilightAutomatic.sObjectName		:= '{Idx=01}';
TwilightAutomatic.eDPADMode			:= E_BA_DPADMode.eInclude;     

ParkPosition.iParent				:= THIS^;	
ParkPosition.iLabel					:= LblCtl_Parking;
ParkPosition.sObjectName			:= '{Idx=01}';
ParkPosition.eDPADMode				:= E_BA_DPADMode.eInclude;     

SunProtection.iParent				:= THIS^;	
SunProtection.iLabel				:= LblCtl_SunProtection;
SunProtection.sObjectName			:= '{Idx=01}';
SunProtection.eDPADMode				:= E_BA_DPADMode.eInclude;     

FacadeInformation.iParent			:= THIS^;	
FacadeInformation.iLabel			:= LblCtl_FacadeInformation;
FacadeInformation.sObjectName		:= '{Idx=01}';
FacadeInformation.eDPADMode			:= E_BA_DPADMode.eInclude;
END_METHOD

END_FUNCTION_BLOCK

// ---- Templates/POUs/Trade/RoomAutomation/SunProtection/Functions/Facade/FB_BA_Facade_WindProtection.TcPOU
{region '#Template'}
	{attribute 'Version' := '5.0.2.0'}
	{attribute 'Tags' := '"LCID": "1031", "Text": "Fassade, Sonnenschutz, Sturmschutz"'}
	{attribute 'Tags' := '"LCID": "1033", "Text": "Facade, Sunprotection, windprotection"'}
	{attribute 'Using' := '"Type": "Template", "URI": "ST_BA_SunBld"'}
	{attribute 'Using' := '"Type": "Template", "URI": "E_BA_SunBldPrio"'}
	{attribute 'Description' := '"LCID": "1031", "Text": "Sturmschutz"'}
	{attribute 'Description' := '"LCID": "1033", "Text": "Windprotection"'}
{endregion}
FUNCTION_BLOCK FB_BA_Facade_WindProtection EXTENDS FB_BA_View
VAR_INPUT
END_VAR
VAR_OUTPUT
	stSunbld					: ST_BA_SunBld;
	bWndPrtc					: BOOL;
	fWndSpdStormOn				: REAL;
	fWndSpdStormOff				: REAL;		
END_VAR
VAR_INPUT CONSTANT PERSISTENT	
	{attribute 'parameterUnit':= 'm/s'}
	aWndSpdLmtStormOn			: ARRAY[1..32] OF REAL;		// Storm-detection on-values for different directions
	{attribute 'parameterUnit':= 'm/s'}
	aWndSpdLmtStormOff			: ARRAY[1..32] OF REAL;		// Storm-detection off-values for different directions
END_VAR
VAR_INPUT CONSTANT
	DlyStrmOn					: FB_BA_AV_Op;		
	DlyStrmOff					: FB_BA_AV_Op;	
	WndPrtcState				: FB_BA_BV_Op;		
	SunBldWndPrtc				: FB_BA_SunBldWndPrtc;
END_VAR
VAR
	aStormDirection				: ARRAY[1..32] OF REAL :=	[0.0, 30.0, 60.0, 90.0, 120.0, 150.0, 180.0, 210.0, 240.0, 270.0, 300.0, 330.0, 360.0];
	StormOnInterpolation		: FB_BA_Chrct32;
	StormOffInterpolation		: FB_BA_Chrct32;
END_VAR

SUPER^(); // FB_BA_View
StormOnInterpolation(
    fX := Site.stWeatherStation.fWindDirection,
    aX := aStormDirection,
    aY := aWndSpdLmtStormOn,
    nNumOfElem := 13); // FB_BA_Chrct32
// Limit ON
fWndSpdStormOn := StormOnInterpolation.fCalcVal;
StormOffInterpolation(
    fX := Site.stWeatherStation.fWindDirection,
    aX := aStormDirection,
    aY := aWndSpdLmtStormOff,
    nNumOfElem := 13); // FB_BA_Chrct32
// Limit OFF
fWndSpdStormOff := StormOffInterpolation.fCalcVal;
// If the resulting value fWndSpdStormOff is bigger than fWndSpdStormOn (by wrong parametrisation), both values shall over the smallest value -> the result is a more sensitive storm-protection
fWndSpdStormOff := MIN(fWndSpdStormOn, fWndSpdStormOff);
DlyStrmOn(); // FB_BA_AV_Op
DlyStrmOff(); // FB_BA_AV_Op
SunBldWndPrtc(
    bEn := TRUE,
    fWndSpd := Site.stWeatherStation.fWindSpeed,
    fWndSpdStrmOn := fWndSpdStormOn,
    fWndSpdStrmOff := fWndSpdStormOff,
    nDlyStrmOn := LIMIT(0, TO_UDINT(DlyStrmOn.fPresentValue), 900),
    nDlyStrmOff := LIMIT(0, TO_UDINT(DlyStrmOff.fPresentValue), 900),
    fPosProt := 0.0,
    fAnglProt := 0.0); // FB_BA_SunBldWndPrtc
stSunbld := SunBldWndPrtc.stSunbld;
WndPrtcState(bValuePgm := SunBldWndPrtc.bActv); // FB_BA_BV_Op
bWndPrtc := WndPrtcState.bPresentValue;

METHOD FB_init : BOOL
VAR_INPUT
	bInitRetains : BOOL; // if TRUE; the retain variables are initialized (warm start / cold start)
	bInCopyCode : BOOL;  // if TRUE; the instance afterwards gets moved into the copy code (online change)
END_VAR
aWndSpdLmtStormOn[01]			:= 12;	// value [m/s] at 0 degree cardinal direction		// default value of 12 is in m/s and means "strong wind" - 6Bft
aWndSpdLmtStormOn[02]			:= 12;	// value [m/s] at 30 degree cardinal direction
aWndSpdLmtStormOn[03]			:= 12;	// value [m/s] at 60 degree cardinal direction
aWndSpdLmtStormOn[04]			:= 12;	// value [m/s] at 90 degree cardinal direction
aWndSpdLmtStormOn[05]			:= 12;	// value [m/s] at 120 degree cardinal direction
aWndSpdLmtStormOn[06]			:= 12;	// value [m/s] at 150 degree cardinal direction
aWndSpdLmtStormOn[07]			:= 12;	// value [m/s] at 180 degree cardinal direction
aWndSpdLmtStormOn[08]			:= 12;	// value [m/s] at 210 degree cardinal direction
aWndSpdLmtStormOn[09]			:= 12;	// value [m/s] at 240 degree cardinal direction
aWndSpdLmtStormOn[10]			:= 12;	// value [m/s] at 270 degree cardinal direction
aWndSpdLmtStormOn[11]			:= 12;	// value [m/s] at 300 degree cardinal direction
aWndSpdLmtStormOn[12]			:= 12;	// value [m/s] at 330 degree cardinal direction
aWndSpdLmtStormOn[13]			:= 12;	// value [m/s] at 360 degree cardinal direction

aWndSpdLmtStormOff[01]			:= 08;	// value [m/s] at 0 degree cardinal direction
aWndSpdLmtStormOff[02]			:= 08;	// value [m/s] at 30 degree cardinal direction
aWndSpdLmtStormOff[03]			:= 08;	// value [m/s] at 60 degree cardinal direction
aWndSpdLmtStormOff[04]			:= 08;	// value [m/s] at 90 degree cardinal direction
aWndSpdLmtStormOff[05]			:= 08;	// value [m/s] at 120 degree cardinal direction
aWndSpdLmtStormOff[06]			:= 08;	// value [m/s] at 150 degree cardinal direction
aWndSpdLmtStormOff[07]			:= 08;	// value [m/s] at 180 degree cardinal direction
aWndSpdLmtStormOff[08]			:= 08;	// value [m/s] at 210 degree cardinal direction
aWndSpdLmtStormOff[09]			:= 08;	// value [m/s] at 240 degree cardinal direction
aWndSpdLmtStormOff[10]			:= 08;	// value [m/s] at 270 degree cardinal direction
aWndSpdLmtStormOff[11]			:= 08;	// value [m/s] at 300 degree cardinal direction
aWndSpdLmtStormOff[12]			:= 08;	// value [m/s] at 330 degree cardinal direction
aWndSpdLmtStormOff[13]			:= 08;	// value [m/s] at 360 degree cardinal direction

DlyStrmOn.iParent				:= THIS^;
DlyStrmOn.iLabel				:= LblCtl_TimeDelayStormOn;
DlyStrmOn.sObjectName			:= '{Idx=01}';
DlyStrmOn.eUnit					:= E_BA_Unit.eTime_Seconds; 
DlyStrmOn.fValueRm				:= 10.0;
                       	
DlyStrmOff.iParent				:= THIS^;
DlyStrmOff.iLabel				:= LblCtl_TimeDelayStormOff;
DlyStrmOff.sObjectName			:= '{Idx=01}';
DlyStrmOff.eUnit				:= E_BA_Unit.eTime_Seconds; 
DlyStrmOff.fValueRm				:= 300.0;
                            	
WndPrtcState.iParent			:= THIS^;	
WndPrtcState.iLabel				:= LblCtl_WindProtectionState;
WndPrtcState.sObjectName		:= '{Idx=01}';
WndPrtcState.sInactiveText		:= txtEvent_Off;
WndPrtcState.sActiveText		:= txtEvent_On;
WndPrtcState.bValueRm			:= FALSE;								
WndPrtcState.eToggleMode 		:= E_BA_ToggleMode.eSwitch;
END_METHOD

END_FUNCTION_BLOCK

// ---- Templates/POUs/Trade/RoomAutomation/SunProtection/Functions/Facade/FB_BA_Facade_Maintenance.TcPOU
{region '#Template'}
	{attribute 'Version' := '5.0.0.0'}
	{attribute 'Tags' := '"LCID": "1031", "Text": "Fassade, Sonnenschutz, Wartung"'}
	{attribute 'Tags' := '"LCID": "1033", "Text": "Facade, Sunprotection, Maintenance"'}
	{attribute 'Using' := '"Type": "Template", "URI": "ST_BA_SunBld"'}
	{attribute 'Using' := '"Type": "Template", "URI": "E_BA_SunBldPrio"'}
	{attribute 'Description' := '"LCID": "1031", "Text": "Sonnenschutz Wartungsposition"'}
	{attribute 'Description' := '"LCID": "1033", "Text": "Sunprotection maintenance-position"'}
{endregion}
FUNCTION_BLOCK FB_BA_Facade_Maintenance EXTENDS FB_BA_View
VAR_INPUT
END_VAR
VAR_OUTPUT
	stSunBld		: ST_BA_SunBld;
	bMntnActv		: BOOL;
END_VAR
VAR_INPUT CONSTANT
	MntnEn			: FB_BA_BV_Op;		
	MntnPos			: FB_BA_AV_Op;		
	MntnAngl		: FB_BA_AV_Op;
	MntnEvent		: FB_BA_SunBldEvt := (ePrio:=E_BA_SunBldPrio.eMaintenance);			
END_VAR
VAR
END_VAR

SUPER^(); // FB_BA_View
MntnEn(); // FB_BA_BV_Op
MntnPos(); // FB_BA_AV_Op
MntnAngl(); // FB_BA_AV_Op
MntnEvent(
    bEn := MntnEn.bPresentValue,
    fPos := LIMIT(0, MntnPos.fPresentValue, 100),
    fAngl := LIMIT(-90, MntnAngl.fPresentValue, 90)); // FB_BA_SunBldEvt
stSunBld := MntnEvent.stSunBld;
bMntnActv := MntnEvent.bActv;

METHOD FB_init : BOOL
VAR_INPUT
	bInitRetains : BOOL; // if TRUE; the retain variables are initialized (warm start / cold start)
	bInCopyCode : BOOL;  // if TRUE; the instance afterwards gets moved into the copy code (online change)
END_VAR
MntnEn.iParent					:= THIS^;
MntnEn.iLabel					:= LblCtl_MaintenanceEnable;
MntnEn.sObjectName		   		:= '{Idx=01}';
MntnEn.sInactiveText			:= txtEvent_Off;
MntnEn.sActiveText				:= txtEvent_On;
MntnEn.bValueRm					:= FALSE;
MntnEn.eToggleMode				:= E_BA_ToggleMode.eSwitch;        
                            	                   	
MntnPos.iParent					:= THIS^;
MntnPos.iLabel					:= LblCtl_MaintenancePosition;
MntnPos.sObjectName		   		:= '{Idx=01}';
MntnPos.eUnit					:= E_BA_Unit.eOther_Percent; 
MntnPos.fValueRm				:= 0.0;
                            	
		                    	
MntnAngl.iParent				:= THIS^;
MntnAngl.iLabel					:= LblCtl_MaintenanceAngle;	
MntnAngl.sObjectName		   	:= '{Idx=02}';
MntnAngl.eUnit					:= E_BA_Unit.eOther_DegreesAngular; 
MntnAngl.fValueRm				:= 0.0;
END_METHOD

END_FUNCTION_BLOCK

// ---- Templates/POUs/Trade/RoomAutomation/SunProtection/Functions/Facade/FB_BA_Facade_ThermoAutomatic.TcPOU
{region '#Template'}
	{attribute 'Version' := '5.0.0.0'}
	{attribute 'Tags' := '"LCID": "1031", "Text": "Fassade, Sonnenschutz, Thermoautomatik"'}
	{attribute 'Tags' := '"LCID": "1033", "Text": "Facade, Sunprotection, thermoautomatic"'}
	{attribute 'Using' := '"Type": "Template", "URI": "ST_BA_SunBld"'}
	{attribute 'Using' := '"Type": "Template", "URI": "E_BA_SunBldPrio"'}
	{attribute 'Description' := '"LCID": "1031", "Text": "Sonnenschutz fassadenweite Thermoautomatik"'}
	{attribute 'Description' := '"LCID": "1033", "Text": "Sunprotection facade-thermoautomatic"'}
{endregion}
FUNCTION_BLOCK FB_BA_Facade_ThermoAutomatic EXTENDS FB_BA_View
VAR_INPUT
	bFcdInSun				: BOOL;	
	fRefRmT					: REAL;
	fRefRmTCol				: REAL;
	fRefRmTHtg				: REAL;	
END_VAR                 	
VAR_OUTPUT              	
	stSunBld				: ST_BA_SunBld;
	bThAutoEvent			: BOOL;
	                    	
END_VAR                 	
VAR_INPUT CONSTANT      	
	FcdThAutoEn				: FB_BA_BV_Op;		
	FcdThAutoColPos			: FB_BA_AV_Op;		
	FcdThAutoColAngl		: FB_BA_AV_Op;		
	FcdThAutoEvent			: FB_BA_SunBldEvt			:=(ePrio:=E_BA_SunBldPrio.eFacadeThermoAutomatic);			
END_VAR                 	
VAR                     	
	FcdThAutoHtgCol			: FB_BA_Swi2P;
	bFcdThAuto_Enable		: BOOL;
	fFcdThAuto_Position		: REAL;
	fFcdThAuto_Angle		: REAL;
END_VAR
VAR // added by the converter: edge detectors and wires of the graphical bodies
    _w1 : BOOL;
END_VAR

SUPER^(); // FB_BA_View
FcdThAutoEn(); // FB_BA_BV_Op
FcdThAutoColPos(); // FB_BA_AV_Op
FcdThAutoColAngl(); // FB_BA_AV_Op
// only if building is not occupied
_w1 := (Site.eBuildingEnergyLevel = E_BA_EnergyLvlEx.eProtection OR Site.eBuildingEnergyLevel = E_BA_EnergyLvlEx.eEconomy) AND Site.stBuildingSunBlind.bGlobalThAuto_Release AND bFcdInSun AND FcdThAutoEn.bPresentValue;
FcdThAutoHtgCol(
    bEn := TRUE,
    fIn := fRefRmT,
    fOn := fRefRmTCol,
    fOff := fRefRmTHtg,
    nDlyOn := 0,
    nDlyOff := 0); // FB_BA_Swi2P
FcdThAutoEvent(
    bEn := _w1,
    fPos := SEL(FcdThAutoHtgCol.bQ, 0, LIMIT(0, FcdThAutoColPos.fPresentValue, 100)),
    fAngl := SEL(FcdThAutoHtgCol.bQ, 0, LIMIT(-90, FcdThAutoColAngl.fPresentValue, 90))); // FB_BA_SunBldEvt
stSunBld := FcdThAutoEvent.stSunBld;
bThAutoEvent := FcdThAutoEvent.bActv;

METHOD FB_init : BOOL
VAR_INPUT
	bInitRetains : BOOL; // if TRUE; the retain variables are initialized (warm start / cold start)
	bInCopyCode : BOOL;  // if TRUE; the instance afterwards gets moved into the copy code (online change)
END_VAR
FcdThAutoEn.iParent				:= THIS^;
FcdThAutoEn.iLabel				:= LblCtl_FacadeThermoAutomaticEnable;
FcdThAutoEn.sObjectName		   	:= '{Idx=01}';
FcdThAutoEn.sInactiveText		:= txtEvent_Off;
FcdThAutoEn.sActiveText			:= txtEvent_On;
FcdThAutoEn.bValueRm			:= FALSE;
FcdThAutoEn.eToggleMode			:= E_BA_ToggleMode.eSwitch;        
                            	
                            	
FcdThAutoColPos.iParent			:= THIS^;  
FcdThAutoColPos.iLabel			:= LblCtl_FacadeThermoAutomaticCoolingPosition;	
FcdThAutoColPos.sObjectName		:= '{Idx=01}';
FcdThAutoColPos.eUnit			:= E_BA_Unit.eOther_Percent; 
FcdThAutoColPos.fValueRm		:= 100.0;
                            	
		                    	
FcdThAutoColAngl.iParent		:= THIS^;
FcdThAutoColAngl.iLabel			:= LblCtl_FacadeThermoAutomaticCoolingAngle;	
FcdThAutoColAngl.sObjectName	:= '{Idx=02}';
FcdThAutoColAngl.eUnit			:= E_BA_Unit.eOther_DegreesAngular; 
FcdThAutoColAngl.fValueRm		:= -90.0;
END_METHOD

END_FUNCTION_BLOCK

// ---- Templates/POUs/Trade/RoomAutomation/SunProtection/Functions/Facade/FB_BA_Facade_ParkPosition.TcPOU
{region '#Template'}
	{attribute 'Version' := '5.0.0.0'}
	{attribute 'Tags' := '"LCID": "1031", "Text": "Fassade, Sonnenschutz, Parkposition"'}
	{attribute 'Tags' := '"LCID": "1033", "Text": "Facade, Sunprotection, parking position"'}
	{attribute 'Using' := '"Type": "Template", "URI": "ST_BA_SunBld"'}
	{attribute 'Using' := '"Type": "Template", "URI": "E_BA_SunBldPrio"'}
	{attribute 'Description' := '"LCID": "1031", "Text": "Sonnenschutz Parkposition"'}
	{attribute 'Description' := '"LCID": "1033", "Text": "Sunprotection parking-position"'}
{endregion}
FUNCTION_BLOCK FB_BA_Facade_ParkPosition EXTENDS FB_BA_View
VAR_INPUT
END_VAR
VAR_OUTPUT
	stSunBld					: ST_BA_SunBld;
	bParkPosEvent				: BOOL;	
END_VAR
VAR_INPUT CONSTANT
	FcdParkEn					: FB_BA_BV_Op;		
	FcdParkPos					: FB_BA_AV_Op;		
	FcdParkAngl					: FB_BA_AV_Op;		
	FcdParkPosEvent				: FB_BA_SunBldEvt :=(ePrio:=E_BA_SunBldPrio.eParkPosition);					
END_VAR
VAR
END_VAR

SUPER^(); // FB_BA_View
FcdParkEn(); // FB_BA_BV_Op
FcdParkPos(); // FB_BA_AV_Op
FcdParkAngl(); // FB_BA_AV_Op
FcdParkPosEvent(
    bEn := FcdParkEn.bPresentValue,
    fPos := LIMIT(0, FcdParkPos.fPresentValue, 100),
    fAngl := LIMIT(-90, FcdParkAngl.fPresentValue, 90)); // FB_BA_SunBldEvt
stSunBld := FcdParkPosEvent.stSunBld;
bParkPosEvent := FcdParkPosEvent.bActv;

METHOD FB_init : BOOL
VAR_INPUT
	bInitRetains : BOOL; // if TRUE; the retain variables are initialized (warm start / cold start)
	bInCopyCode : BOOL;  // if TRUE; the instance afterwards gets moved into the copy code (online change)
END_VAR
FcdParkEn.iParent				:= THIS^;
FcdParkEn.iLabel				:= LblCtl_FacadeParkingEnable;
FcdParkEn.sObjectName			:= '{Idx=01}';
FcdParkEn.sInactiveText			:= txtEvent_Off;
FcdParkEn.sActiveText			:= txtEvent_On;
FcdParkEn.bValueRm				:= FALSE;
FcdParkEn.eToggleMode			:= E_BA_ToggleMode.eSwitch;        

FcdParkPos.iParent				:= THIS^;
FcdParkPos.iLabel				:= LblCtl_FacadeParkingPosition;
FcdParkPos.sObjectName			:= '{Idx=01}';
FcdParkPos.eUnit				:= E_BA_Unit.eOther_Percent; 
FcdParkPos.fValueRm				:= 0.0;
FcdParkPos.fCOVIncrement		:= BA2_Param.fDefCOVIncrement;
		  
FcdParkAngl.iParent				:= THIS^;
FcdParkAngl.iLabel				:= LblCtl_FacadeParkingAngle;
FcdParkAngl.sObjectName			:= '{Idx=02}';
FcdParkAngl.eUnit				:= E_BA_Unit.eOther_DegreesAngular; 
FcdParkAngl.fValueRm			:= 0.0; 
FcdParkAngl.fCOVIncrement		:= BA2_Param.fDefCOVIncrement;
END_METHOD

END_FUNCTION_BLOCK

// ---- Templates/POUs/Trade/RoomAutomation/SunProtection/Functions/Facade/FB_BA_Facade_Information.TcPOU
{region '#Template'}
	{attribute 'Version' := '5.0.0.0'}
	{attribute 'Tags' := '"LCID": "1031", "Text": "Fassade, Sonnenschutz, Parkposition"'}
	{attribute 'Tags' := '"LCID": "1033", "Text": "Facade, Sunprotection, parking position"'}
	{attribute 'Using' := '"Type": "Template", "URI": "ST_BA_SunBld"'}
	{attribute 'Using' := '"Type": "Template", "URI": "E_BA_SunBldPrio"'}
	{attribute 'Description' := '"LCID": "1031", "Text": "Sonnenschutz Parkposition"'}
	{attribute 'Description' := '"LCID": "1033", "Text": "Sunprotection parking-position"'}
{endregion}
FUNCTION_BLOCK FB_BA_Facade_Information EXTENDS FB_BA_View
VAR_INPUT
	stFacadeResult				: ST_BA_SunBld;
END_VAR
VAR_INPUT CONSTANT
	FcdActvPrio					: FB_BA_MV_Op;			
END_VAR

SUPER^(); // FB_BA_View
FcdActvPrio(nValuePgm := stFacadeResult.ePrio + 1); // FB_BA_MV_Op

METHOD FB_init : BOOL
VAR_INPUT
	bInitRetains : BOOL; // if TRUE; the retain variables are initialized (warm start / cold start)
	bInCopyCode : BOOL;  // if TRUE; the instance afterwards gets moved into the copy code (online change)
END_VAR

FcdActvPrio.iParent				:= THIS^;
FcdActvPrio.iLabel				:= LblCtl_PrioResultingTelegram;
FcdActvPrio.aStateText[1]		:= txtEvent_None;
FcdActvPrio.aStateText[2]		:= txtEvent_Fire;
FcdActvPrio.aStateText[3]		:= txtEvent_Storm;
FcdActvPrio.aStateText[4]		:= txtEvent_Ice;
FcdActvPrio.aStateText[5]		:= txtEvent_CommError;
FcdActvPrio.aStateText[6]		:= txtEvent_Burglary;
FcdActvPrio.aStateText[7]		:= txtEvent_Maintenance;
FcdActvPrio.aStateText[8]		:= txtEvent_Referencing;
FcdActvPrio.aStateText[9]		:= txtEvent_ManualActuator;
FcdActvPrio.aStateText[10]   	:= txtEvent_ManualGroup;
FcdActvPrio.aStateText[11]		:= txtEvent_AllDown;
FcdActvPrio.aStateText[12]		:= txtEvent_AllUp;	              
FcdActvPrio.aStateText[13]		:= txtEvent_Scene1;            
FcdActvPrio.aStateText[14]		:= txtEvent_FacadeThermoAutomatic;
FcdActvPrio.aStateText[15]		:= txtEvent_FacadeTwilightAutomatic;
FcdActvPrio.aStateText[16]		:= txtEvent_ParkPosition;
FcdActvPrio.aStateText[17]		:= txtEvent_Scene2;
FcdActvPrio.aStateText[18]		:= txtEvent_Scene3;
FcdActvPrio.aStateText[19]		:= txtEvent_SunProtection;
FcdActvPrio.aStateText[20]		:= txtEvent_GroupThermoAuto;
FcdActvPrio.aStateText[21]		:= txtEvent_GroupTwiLightAuto;
END_METHOD

END_FUNCTION_BLOCK

// ---- Templates/POUs/Trade/AirConditioning/Aggregates/Cooler/Temperature/FB_BA_AC_ColTSuACtrl.TcPOU
{region '#Template'}
	{attribute 'Version' := '5.0.1.0'}
	{attribute 'Tags' := '"LCID": "1031", "Text": "AC, Aggregates, Cooler, Temperature, Controller"'}
	{attribute 'Tags' := '"LCID": "1033", "Text": "AC, Aggregates, Cooler, Temperature, Controller"'}
	{attribute 'Using' := '"Type": "Template", "URI": "BA2_Param"'}
	{attribute 'Using' := '"Type": "Template", "URI": "EC_ID"'}
	{attribute 'Using' := '"Type": "Template", "URI": "E_BA_AC_SeqNumber_T"'}
	{attribute 'Description' := '"LCID": "1031", "Text": "Kühler Zuluft Regler Temperatur"'}
	{attribute 'Description' := '"LCID": "1033", "Text": "Cooler Supply air controller temperature"'}
{endregion}
FUNCTION_BLOCK FB_BA_AC_ColTSuACtrl EXTENDS FB_BA_View
VAR_INPUT
	bEn						: BOOL;
	fSpTSuA					: REAL;// Sollwert Temperatur kühlen // Setpoint temperature cooling
	fTSuA					: REAL;// Zuluft Temperatur // Supply air temperature
	bSync					: BOOL;
	fSync					: REAL;
END_VAR
VAR_OUTPUT
	fY              		: REAL;
	bIsActive				: BOOL;	//	active sequence controller
	bSeqActv				: BOOL;	//	Release sequence link, sequence control is active		
END_VAR
VAR_IN_OUT
	stSeqLink				: ST_BA_SeqLink;	//	Sequenz Link Struktur	//	Sequence link structure	
END_VAR
VAR_INPUT CONSTANT
	Ctrl					: FB_BA_SeqCtrl;
END_VAR

SUPER^(); // FB_BA_View
Ctrl(
    bEn := bEn AND stSeqLink.bEnSeqLink,
    fSetpoint := fSpTSuA,
    fCtrlVal := fTSuA,
    eActionPgm := E_BA_Action.eDirect,
    bEnSync := bSync,
    fValSync := fSync,
    nMyNum := E_BA_AC_SeqNumber_T.eCooler,
    stSeqLink := stSeqLink); // FB_BA_SeqCtrl
fY := Ctrl.fPresentValue;
bSeqActv := Ctrl.bSeqActv;
bIsActive := Ctrl.bIsActvSeqCtrl;

METHOD FB_init : BOOL
VAR_INPUT
	bInitRetains : BOOL; // if TRUE, the retain variables are initialized (warm start / cold start)
	bInCopyCode : BOOL;  // if TRUE, the instance afterwards gets moved into the copy code (online change)
END_VAR
Ctrl.iParent						:= THIS^;
Ctrl.iLabel							:= LblFun_LoopObject; 
Ctrl.sObjectName					:= '{Idx=01}';						 
Ctrl.eOpMode						:= E_BA_PIDMode.ePID;								 	 										 	
Ctrl.eOutputUnit					:= E_BA_Unit.eOther_Percent;
Ctrl.fProportionalConstant			:= 3;
Ctrl.fIntegralConstant				:= 180;
Ctrl.fDerivativeConstant			:= 0;
Ctrl.fMaxOutputRm 					:= 100;
Ctrl.fMinOutputRm					:= 0;
Ctrl.fCOVIncrement					:= 0;
Ctrl.nDampConstant					:= 0;
Ctrl.fNeutralZone					:= 0;
END_METHOD

END_FUNCTION_BLOCK

// ---- Templates/POUs/Trade/AirConditioning/Aggregates/Cooler/Temperature/FB_BA_AC_ColT_02.TcPOU
{region '#Template'}
	{attribute 'Version' := '6.0.0.0'}
	{attribute 'Tags' := '"LCID": "1031", "Text": "AC, Aggregates, Cooler, Temperature"'}
	{attribute 'Tags' := '"LCID": "1033", "Text": "AC, Aggregates, Cooler, Temperature"'}
	{attribute 'Using' := '"Type": "Template", "URI": "Priority"'}		 		 
	{attribute 'Description' := '"LCID": "1031", "Text": "Aggregat Kühler Temperatur mit Ventil"'}
	{attribute 'Description' := '"LCID": "1033", "Text": "Aggregate cooler temperature with valve"'}
{endregion}
FUNCTION_BLOCK FB_BA_AC_ColT_02 EXTENDS FB_BA_View
VAR_INPUT
	fSpTSuA					: REAL;// Sollwert Temperatur kühlen // Setpoint temperature cooling
	fTSuA					: REAL;// Zuluft Temperatur // Supply air temperature
	bSyncTSuACtrl			: BOOL;
	fSyncTSuACtrl			: REAL;		
END_VAR
VAR_OUTPUT
	fPresentValue			: REAL;	
	bActiveSeqCtrl			: BOOL;
END_VAR
VAR_IN_OUT
	stTSeqLink				: ST_BA_SeqLink;	//	Sequenz Link Struktur	//	Sequence link structure	
	stAggregate				: ST_BA_Aggregate;	
END_VAR
VAR_INPUT CONSTANT
	TFl						: FB_BA_SensorAnalog;												
	TRt						: FB_BA_SensorAnalog;			
	TSuACtrl				: FB_BA_AC_ColTSuACtrl;
	Vlv						: FB_BA_Vlv;
	PlantLock				: FB_BA_PlantLock;																							
	Aggregate				: FB_BA_Aggregate;	
END_VAR
VAR		
	bPrioSfty				: BOOL;
	bPrioCrit				: BOOL;		
	PrioSwiVal				: FB_BA_PrioSwi_B04;	
END_VAR
VAR // added by the converter: edge detectors and wires of the graphical bodies
    _s1 : ST_BA_Analog;
END_VAR

SUPER^(); // FB_BA_View
Aggregate(stAggregate := stAggregate); // FB_BA_Aggregate
PlantLock(); // FB_BA_PlantLock
bPrioSfty := PlantLock.bPrioHigh OR PlantLock.bPrioLocalHigh;
bPrioCrit := PlantLock.bPrioMedium OR PlantLock.bPrioLocalMedium;
TFl(); // FB_BA_SensorAnalog
TRt(); // FB_BA_SensorAnalog
PrioSwiVal(
    bEn01 := Aggregate.arrPriorities[Priority.nLifeSafety],
    bVal01 := Aggregate.bValue,
    bEn02 := Aggregate.arrPriorities[Priority.nCritical],
    bVal02 := Aggregate.bValue,
    bEn03 := Aggregate.arrPriorities[Priority.nProgram],
    bVal03 := Aggregate.bValue); // FB_BA_PrioSwi_B04
TSuACtrl(
    bEn := PrioSwiVal.bVal,
    fSpTSuA := fSpTSuA,
    fTSuA := fTSuA,
    bSync := bSyncTSuACtrl,
    fSync := fSyncTSuACtrl,
    stSeqLink := stTSeqLink); // FB_BA_AC_ColTSuACtrl
bActiveSeqCtrl := TSuACtrl.bIsActive;
// compose _s1 : ST_BA_Analog
_s1.bEnSfty := Aggregate.arrPriorities[Priority.nLifeSafety] OR bPrioSfty;
_s1.fValSfty := TSuACtrl.fY;
_s1.bEnCrit := Aggregate.arrPriorities[Priority.nCritical] OR bPrioCrit;
_s1.fValCrit := TSuACtrl.fY;
_s1.bEnPgm := Aggregate.arrPriorities[Priority.nProgram];
_s1.fValPgm := TSuACtrl.fY;
Vlv(stCmd := _s1); // FB_BA_Vlv
fPresentValue := Vlv.fMdlt;

METHOD FB_init : BOOL
VAR_INPUT
	bInitRetains : BOOL; // if TRUE, the retain variables are initialized (warm start / cold start)
	bInCopyCode : BOOL;  // if TRUE, the instance afterwards gets moved into the copy code (online change)
END_VAR
PlantLock.Parent								:= THIS^;		

TFl.iParent								:= THIS^;		
TFl.iLabel								:= LblAgg_TemperatureFlow;   
TFl.sObjectName							:= '{Idx=41}';						 
TFl.eDPADMode							:= E_BA_DPADMode.eInclude;															
TFl.MV.eUnit							:= E_BA_Unit.eTemperature_DegreesCelsius;
TFl.MV.fResolution 						:= 0.01;
TFl.MV.fScaleOffset 					:= 0; 
TFl.MV.bEventDetectionEnable			:= TRUE;
TFl.MV.eEnPlantLock						:= E_BA_LockPriority.eNoLock;

TRt.iParent								:= THIS^;		
TRt.iLabel								:= LblAgg_TemperatureReturnFlow;
TRt.sObjectName							:= '{Idx=41}';						 
TRt.eDPADMode							:= E_BA_DPADMode.eInclude;																												
TRt.MV.eUnit							:= E_BA_Unit.eTemperature_DegreesCelsius;
TRt.MV.fResolution 						:= 0.01;
TRt.MV.fScaleOffset 					:= 0;  
TRt.MV.bEventDetectionEnable			:= TRUE;	
TRt.MV.eEnPlantLock						:= E_BA_LockPriority.eNoLock;

TSuACtrl.iParent						:= THIS^;	 
TSuACtrl.iLabel							:= LblCtl_SupplyAirTemperatureControl;
TSuACtrl.sObjectName					:= '{Idx=41}';						 
TSuACtrl.eDPADMode						:= E_BA_DPADMode.eInclude;								
                        				
Vlv.iParent								:= THIS^;
Vlv.iLabel								:= LblAgg_Valve;
Vlv.sObjectName							:= '{Idx=41}';						 
Vlv.eDPADMode							:= E_BA_DPADMode.eInclude;
END_METHOD

END_FUNCTION_BLOCK

// ---- Templates/POUs/Universal/Valve/FB_BA_Vlv.TcPOU
{region '#Template'}
	{attribute 'Version' := '5.0.0.0'}
	{attribute 'Tags' := '"LCID": "1031", "Text": "Universal, Valve"'}
	{attribute 'Tags' := '"LCID": "1033", "Text": "Universal, Valve"'}
	{attribute 'Using' := '"Type": "Template", "URI": "EC_ID"'}
	{attribute 'Using' := '"Type": "Template", "URI": "BA2_Param"'}
	{attribute 'Description' := '"LCID": "1031", "Text": "Ventil analog"'}
	{attribute 'Description' := '"LCID": "1033", "Text": "Valve analog"'}
{endregion}		 
FUNCTION_BLOCK FB_BA_Vlv EXTENDS FB_BA_ActuatorAnalog
VAR_INPUT
	bAblkLock				: BOOL;
END_VAR
VAR_OUTPUT
END_VAR
VAR_INPUT CONSTANT
	Ablk					: FB_BA_AntiBlocking;	
	Fdb						: FB_BA_AI_Raw;		 
END_VAR
VAR // added by the converter: edge detectors and wires of the graphical bodies
    _s1 : ST_BA_Analog;
END_VAR

Fdb(); // FB_BA_AI_Raw
Ablk(bFdb := fMdlt >= 30.0, bLock := bAblkLock); // FB_BA_AntiBlocking
// compose _s1 : ST_BA_Analog
_s1.bEnSfty := stCmd.bEnSfty;
_s1.fValSfty := stCmd.fValSfty;
_s1.bEnCrit := stCmd.bEnCrit;
_s1.fValCrit := stCmd.fValCrit;
_s1.bEnPgm := Ablk.bQ OR stCmd.bEnPgm;
_s1.fValPgm := SEL(Ablk.bQ, stCmd.fValPgm, 100);
SUPER^(stCmd := _s1); // FB_BA_ActuatorAnalog

METHOD FB_init : BOOL
VAR_INPUT
	bInitRetains : BOOL; // if TRUE, the retain variables are initialized (warm start / cold start)
	bInCopyCode : BOOL;  // if TRUE, the instance afterwards gets moved into the copy code (online change)
END_VAR
Ablk.iParent					:= THIS^;	
Ablk.iLabel						:= LblCtl_AntiBlocking;  
Ablk.eDPADMode					:= E_BA_DPADMode.eIncludeDescription;

Fdb.iParent						:= THIS^;		
Fdb.iLabel						:= LblFun_Feedback;  
Fdb.eUnit						:= E_BA_Unit.eOther_Percent;
Fdb.fResolution 				:= 0.03051851;
Fdb.fScaleOffset 				:= 0; 	
Fdb.fCOVIncrement				:= BA2_Param.fDefCOVIncrement;
Fdb.nEventClassID				:= EC_ID.NC80;
Fdb.stTimeDelay.nToNormal		:= BA2_Param.nDefTimeDelay_ToNormal;
Fdb.stTimeDelay.nToAbnormal		:= BA2_Param.nDefTimeDelay_ToAbnormal;
Fdb.stHighLimit.bEnable			:= FALSE;
Fdb.stHighLimit.fValue			:= 0.0;		
Fdb.stLowLimit.bEnable			:= FALSE;
Fdb.stLowLimit.fValue			:= 0.0;
Fdb.fLimitDeadband 				:= BA2_Param.fDefLimitDeadband;
Fdb.aEventTransitionText[1]		:= txtEvent_Exceeded;
Fdb.aEventTransitionText[2]		:= txtEvent_Disturb;
Fdb.aEventTransitionText[3]		:= txtEvent_Normal;
Fdb.bEventDetectionEnable		:= FALSE;
Fdb.eEnPlantLock				:= E_BA_LockPriority.eNoLock;
END_METHOD

END_FUNCTION_BLOCK

// ---- Templates/POUs/Universal/Control/AntiBlocking/FB_BA_AntiBlocking.TcPOU
{region '#Template'}
	{attribute 'Version' := '5.0.0.0'}
	{attribute 'Tags' := '"LCID": "1031", "Text": "Universal, Control, Antiblockierschutz"'}
	{attribute 'Tags' := '"LCID": "1033", "Text": "Universal, Control, Anti-blocking protection"'}
	{attribute 'Using' := '"Type": "Template", "URI": "EC_ID"'}
	{attribute 'Using' := '"Type": "Template", "URI": "BA2_Param"'}
	{attribute 'Description' := '"LCID": "1031", "Text": "Antiblockierschutz"'}
	{attribute 'Description' := '"LCID": "1033", "Text": "Anti-blocking protection"'}
{endregion}
FUNCTION_BLOCK FB_BA_AntiBlocking EXTENDS FB_BA_View
VAR_INPUT
	bFdb					: BOOL;	
	bExtReq					: BOOL;
	bLock					: BOOL;
END_VAR
VAR_OUTPUT
	bQ						: BOOL;
END_VAR
VAR_INPUT CONSTANT PERSISTENT
	{attribute 'parameterCategory' := 'Operation'}
	bEn : BOOL := TRUE;
END_VAR
VAR_INPUT CONSTANT
	IdlePrd					: FB_BA_AV_Op;									 
	ImpulseLength			: FB_BA_AV_Op;
END_VAR	
VAR		
	AblkFnct				: FB_BA_AntBlkg;
	tonEn					: TON;
END_VAR

SUPER^(); // FB_BA_View
IdlePrd(); // FB_BA_AV_Op
AblkFnct.nOffMin := MAX(TO_UDINT(IdlePrd.fPresentValue) * 3600, 60);
ImpulseLength(); // FB_BA_AV_Op
AblkFnct.nImplLngt := MAX(TO_UDINT(ImpulseLength.fPresentValue), 10);
AblkFnct(bEn := bEn AND BA2_Param.bDlyStartPLC, bFdb := bFdb, bExtReq := bExtReq, bLock := bLock); // FB_BA_AntBlkg
bQ := AblkFnct.bQ;

METHOD FB_init : BOOL
VAR_INPUT
	bInitRetains : BOOL; // if TRUE, the retain variables are initialized (warm start / cold start)
	bInCopyCode : BOOL;  // if TRUE, the instance afterwards gets moved into the copy code (online change)
END_VAR
IdlePrd.iParent					:= THIS^; 
IdlePrd.iLabel					:= LblCtl_IdlePeriod;								 	 
IdlePrd.eUnit 					:= E_BA_Unit.eTime_Hours;								 
IdlePrd.fValueRm				:= 168;
IdlePrd.fCOVIncrement			:= BA2_Param.fDefCOVIncrement;
														 
ImpulseLength.iParent			:= THIS^;
ImpulseLength.iLabel			:= LblCtl_ImpulsLength;									 	 
ImpulseLength.eUnit 			:= E_BA_Unit.eTime_Seconds;								 
ImpulseLength.fValueRm			:= 240;					
ImpulseLength.fCOVIncrement		:= BA2_Param.fDefCOVIncrement;
END_METHOD

END_FUNCTION_BLOCK

// ---- Templates/POUs/Trade/AirConditioning/Aggregates/Damper/FB_BA_AC_Dmp2P.TcPOU
{region '#Template'}
	{attribute 'Version' := '6.0.0.0'}
	{attribute 'Tags' := '"LCID": "1031", "Text": "AC, Aggregate, Klappe"'}
	{attribute 'Tags' := '"LCID": "1033", "Text": "AC, Aggregate, Damper"'}
	{attribute 'Using' := '"Type": "Template", "URI": "Priority"'}		 
	{attribute 'Using' := '"Type": "Template", "URI": "EC_ID"'}
	{attribute 'Using' := '"Type": "Template", "URI": "BA2_Param"'}
	{attribute 'Description' := '"LCID": "1031", "Text": "2 Punkt Klappe mit Endlagenschalter"'}
	{attribute 'Description' := '"LCID": "1033", "Text": "2 point damper with limit switch"'}
{endregion}			 
FUNCTION_BLOCK FB_BA_AC_Dmp2P EXTENDS FB_BA_ActuatorCmd
VAR_INPUT
	bFan					: BOOL;
END_VAR
VAR_OUTPUT
	bSwiOpn					: BOOL;
	bSwiCls					: BOOL;
END_VAR
VAR_IN_OUT
	stAggregate				: ST_BA_Aggregate;	
END_VAR
VAR_INPUT CONSTANT
	SwiOpn					: FB_BA_BI_Raw;
	SwiCls					: FB_BA_BI_Raw;
	MonitOpen				: FB_BA_FdbBinary;
	MonitClose				: FB_BA_FdbBinary;
	Aggregate				: FB_BA_Aggregate;																											 							
END_VAR	
VAR	
	PrioSwiFan				: FB_BA_PrioSwi_B04;
END_VAR
VAR // added by the converter: edge detectors and wires of the graphical bodies
    _s1 : ST_BA_Binary;
END_VAR

Aggregate(bFdbUp := bSwiOpn, bFdbDown := bSwiCls, stAggregate := stAggregate); // FB_BA_Aggregate
SwiOpn(); // FB_BA_BI_Raw
bSwiOpn := SwiOpn.bPresentValue;
SwiCls(); // FB_BA_BI_Raw
bSwiCls := SwiCls.bPresentValue;
PrioSwiFan(
    bEn01 := bFan,
    bVal01 := TRUE,
    bEn03 := Aggregate.arrPriorities[Priority.nCritical],
    bVal03 := Aggregate.bValue); // FB_BA_PrioSwi_B04
// compose _s1 : ST_BA_Binary
_s1.bEnSfty := Aggregate.arrPriorities[Priority.nLifeSafety];
_s1.bValSfty := Aggregate.bValue;
_s1.bEnCrit := PrioSwiFan.bQ;
_s1.bValCrit := PrioSwiFan.bVal;
_s1.bEnPgm := Aggregate.arrPriorities[Priority.nProgram];
_s1.bValPgm := Aggregate.bValue;
SUPER^(stCmd := _s1); // FB_BA_ActuatorCmd
MonitOpen(bEn := BA2_Param.bDlyStartPLC, bCommand := bCmd, bFeedback := bSwiOpn); // FB_BA_FdbBinary
MonitClose(bEn := BA2_Param.bDlyStartPLC, bCommand := NOT bCmd, bFeedback := bSwiCls); // FB_BA_FdbBinary

METHOD FB_init : BOOL
VAR_INPUT
	bInitRetains : BOOL; // if TRUE, the retain variables are initialized (warm start / cold start)
	bInCopyCode : BOOL;  // if TRUE, the instance afterwards gets moved into the copy code (online change)
END_VAR
SwiOpn.iParent							:= THIS^;
SwiOpn.iLabel							:= LblFun_FeedbackOPEN;  
SwiOpn.sObjectName						:='{Idx=01}';
SwiOpn.ePolarity						:= E_BA_Polarity.eReverse;
SwiOpn.sActiveText 						:= txtEvent_Reached;
SwiOpn.sInactiveText 					:= txtEvent_NotReached;
SwiOpn.nEventClassID					:= EC_ID.NC80;
SwiOpn.stTimeDelay.nToNormal			:= BA2_Param.nDefTimeDelay_ToNormal;
SwiOpn.stTimeDelay.nToAbnormal			:= BA2_Param.nDefTimeDelay_ToAbnormal;
SwiOpn.bAlarmValue						:= TRUE;
SwiOpn.aEventTransitionText[1]			:= txtEvent_Active;
SwiOpn.aEventTransitionText[2]			:= txtEvent_None;
SwiOpn.aEventTransitionText[3]			:= txtEvent_Normal;
SwiOpn.bEventDetectionEnable			:= FALSE;
SwiOpn.eEnPlantLock						:= E_BA_LockPriority.eNoLock;	

SwiCls.iParent							:= THIS^;
SwiCls.iLabel							:= LblFun_FeedbackCLOSED; 
SwiCls.sObjectName						:='{Idx=01}';
SwiCls.ePolarity						:= E_BA_Polarity.eReverse;
SwiCls.sActiveText 						:= txtEvent_Reached;
SwiCls.sInactiveText 					:= txtEvent_NotReached;
SwiCls.nEventClassID					:= EC_ID.NC80;
SwiCls.stTimeDelay.nToNormal			:= BA2_Param.nDefTimeDelay_ToNormal;
SwiCls.stTimeDelay.nToAbnormal			:= BA2_Param.nDefTimeDelay_ToAbnormal;
SwiCls.bAlarmValue						:= TRUE;
SwiCls.aEventTransitionText[1]			:= txtEvent_Active;
SwiCls.aEventTransitionText[2]			:= txtEvent_None;
SwiCls.aEventTransitionText[3]			:= txtEvent_Normal;
SwiCls.bEventDetectionEnable			:= FALSE;
SwiCls.eEnPlantLock						:= E_BA_LockPriority.eNoLock;

MonitOpen.iParent						:= THIS^;
MonitOpen.iLabel						:= LblCtl_FeedbackMonitoring;  
MonitOpen.sObjectName					:='{Idx=01}';
MonitOpen.eDPADMode						:= E_BA_DPADMode.eIncludeDescription;
MonitOpen.DelayFeedback.fValueRm		:= 180.0;
MonitOpen.DelayFeedback.sObjectName		:='{Idx=01}';
MonitOpen.Dst.bEventDetectionEnable		:= TRUE;
MonitOpen.Dst.eEnPlantLock				:= E_BA_LockPriority.eLocalMedium;

MonitClose.iParent						:= THIS^;
MonitClose.iLabel						:= LblCtl_FeedbackMonitoring;
MonitClose.sObjectName					:='{Idx=02}';
MonitClose.eDPADMode					:= E_BA_DPADMode.eIncludeDescription;
MonitClose.DelayFeedback.fValueRm		:= 180.0;
MonitClose.DelayFeedback.iLabel			:= LblFun_FeedbackDelay;
MonitClose.DelayFeedback.sObjectName	:='{Idx=02}';
MonitClose.Dst.iLabel					:= LblFun_Fault;
MonitClose.Dst.sObjectName				:='{Idx=02}';
MonitClose.Dst.bEventDetectionEnable	:= TRUE;
MonitClose.Dst.eEnPlantLock				:= E_BA_LockPriority.eNoLock;
END_METHOD

END_FUNCTION_BLOCK

// ---- Templates/POUs/Universal/Control/Monitoring/FB_BA_FdbBinary.TcPOU
{region '#Template'}
	{attribute 'Version' := '5.0.0.0'}
	{attribute 'Tags' := '"LCID": "1031", "Text": "Universal, Control, Monitoring"'}
	{attribute 'Tags' := '"LCID": "1033", "Text": "Universal, Control, Monitoring"'}
	{attribute 'Using' := '"Type": "Template", "URI": "EC_ID"'}
	{attribute 'Using' := '"Type": "Template", "URI": "BA2_Param"'}
	{attribute 'Description' := '"LCID": "1031", "Text": "Überwachung von Signalen"'}
	{attribute 'Description' := '"LCID": "1033", "Text": "Monitoring signals"'}
{endregion}
FUNCTION_BLOCK FB_BA_FdbBinary EXTENDS FB_BA_View
VAR_INPUT
	bEn						: BOOL;	
	bCommand				: BOOL;	
	bFeedback				: BOOL;		
END_VAR
VAR_OUTPUT
	bDst					: BOOL;
END_VAR
VAR_INPUT CONSTANT
	DelayFeedback			: FB_BA_AV_Op;
	Dst						: FB_BA_BV;			
END_VAR
VAR_INPUT CONSTANT PERSISTENT
	{attribute 'parameterUnit':= 's'}
	nInterruptionDelay : UDINT := 1;
END_VAR
VAR
	FdbCtrl					: FB_BA_FdbCtrlBinary;		
END_VAR

SUPER^(); // FB_BA_View
DelayFeedback(); // FB_BA_AV_Op
FdbCtrl(
    bEn := bEn,
    bActuator := bCommand,
    bSwitch := bFeedback,
    nFdbDelay := TO_UDINT(DelayFeedback.fPresentValue),
    nInterruptionDelay := nInterruptionDelay); // FB_BA_FdbCtrlBinary
Dst(bEnPgm := TRUE, bValPgm := FdbCtrl.bQ); // FB_BA_BV
bDst := Dst.bEvent;

METHOD FB_init : BOOL
VAR_INPUT
	bInitRetains : BOOL; // if TRUE, the retain variables are initialized (warm start / cold start)
	bInCopyCode : BOOL;  // if TRUE, the instance afterwards gets moved into the copy code (online change)
END_VAR
DelayFeedback.iParent				:= THIS^;
DelayFeedback.iLabel				:= LblFun_FeedbackDelay;	 	 
DelayFeedback.eUnit 				:= E_BA_Unit.eTime_Seconds;								 
DelayFeedback.fValueRm 				:= 120;
DelayFeedback.fCOVIncrement			:= BA2_Param.fDefCOVIncrement;		

Dst.iParent							:= THIS^;
Dst.iLabel							:= LblFun_Fault;
Dst.sActiveText 					:= txtEvent_Triggered;
Dst.sInactiveText 					:= txtEvent_Normal;
Dst.bEnManualRm						:= FALSE;	//	Priority  8	
Dst.bValManualRm					:= FALSE;	//	Priority  8
Dst.nEventClassID					:= EC_ID.NC30;
Dst.stTimeDelay.nToNormal			:= 0;
Dst.stTimeDelay.nToAbnormal			:= 0;
Dst.bAlarmValue						:= TRUE;
Dst.aEventTransitionText[1]			:= txtEvent_Triggered;
Dst.aEventTransitionText[2]			:= txtEvent_Error;
Dst.aEventTransitionText[3]			:= txtEvent_Normal;
Dst.bEventDetectionEnable			:= TRUE;
Dst.eEnPlantLock					:= E_BA_LockPriority.eNoLock;
END_METHOD

END_FUNCTION_BLOCK

// ---- Templates/POUs/Trade/AirConditioning/Aggregates/ERC/FB_BA_AC_ErcTSuACtrl.TcPOU
{region '#Template'}
	{attribute 'Version' := '5.0.1.0'}
	{attribute 'Tags' := '"LCID": "1031", "Text": "AC, Aggregates, Energy recovery, Temperature, Controller"'}
	{attribute 'Tags' := '"LCID": "1033", "Text": "AC, Aggregates, Energy recovery, Temperature, Controller"'}
	{attribute 'Using' := '"Type": "Template", "URI": "BA2_Param"'}
	{attribute 'Using' := '"Type": "Template", "URI": "EC_ID"'}
	{attribute 'Using' := '"Type": "Template", "URI": "E_BA_AC_SeqNumber_T"'}		 
	{attribute 'Description' := '"LCID": "1031", "Text": "Energie Rückgewinnung Zuluft Regler Temperatur"'}
	{attribute 'Description' := '"LCID": "1033", "Text": "Energy recovery Supply air controller temperature"'}
{endregion}
FUNCTION_BLOCK FB_BA_AC_ErcTSuACtrl EXTENDS FB_BA_View
VAR_INPUT
	bEn					: BOOL;
	fSpTSuA				: REAL;
	fTSuA				: REAL;
	bSync				: BOOL;
	fSync				: REAL;
	bDehumf				: BOOL;
	fTExtA				: REAL;
	fTWth				: REAL;
END_VAR
VAR_OUTPUT
	fY					: REAL;
	eAction				: E_BA_Action;
	bIsActive				: BOOL;	//	active sequence controller
	bSeqActv				: BOOL;	//	Release sequence link, sequence control is active	
END_VAR
VAR_IN_OUT
	stSeqLink			: ST_BA_SeqLink;	//	Sequenz Link Struktur	//	Sequence link structure	
END_VAR
VAR_INPUT CONSTANT PERSISTENT
	{attribute 'parameterCategory' := 'Behaviour'}
	fHysActionOn 		: REAL := 0.25;
	{attribute 'parameterCategory' := 'Behaviour'}
	fHysActionOff 		: REAL := -0.25;
END_VAR
VAR_INPUT CONSTANT
	Ctrl				: FB_BA_SeqCtrl;		 
END_VAR
VAR		
	HysAction			: FB_BA_Swi2P;
END_VAR

SUPER^(); // FB_BA_View
HysAction(bEn := TRUE, fIn := fTWth - fTExtA, fOn := fHysActionOn, fOff := fHysActionOff); // FB_BA_Swi2P
Ctrl(
    fSetpoint := fSpTSuA,
    fCtrlVal := fTSuA,
    eActionPgm := SEL(HysAction.bQ, E_BA_Action.eReverse, E_BA_Action.eDirect),
    bEnSync := bSync,
    fValSync := fSync,
    bEn := bEn AND NOT (bDehumf AND eAction = E_BA_Action.eReverse),
    nMyNum := E_BA_AC_SeqNumber_T.eEnergyRecovery,
    stSeqLink := stSeqLink); // FB_BA_SeqCtrl
fY := Ctrl.fPresentValue;
bSeqActv := Ctrl.bSeqActv;
bIsActive := Ctrl.bIsActvSeqCtrl;
eAction := Ctrl.Actn;

METHOD FB_init : BOOL
VAR_INPUT
	bInitRetains : BOOL; // if TRUE, the retain variables are initialized (warm start / cold start)
	bInCopyCode : BOOL;  // if TRUE, the instance afterwards gets moved into the copy code (online change)
END_VAR
Ctrl.iParent						:= THIS^;
Ctrl.iLabel							:= LblFun_LoopObject; 		
Ctrl.sObjectName					:= '{Idx=01}';						 
Ctrl.eOpMode						:= E_BA_PIDMode.ePID;								 	 										 
Ctrl.eOutputUnit					:= E_BA_Unit.eOther_Percent;
Ctrl.eActionRm						:= E_BA_Action.eReverse;
Ctrl.fProportionalConstant			:= 3;
Ctrl.fIntegralConstant				:= 180;
Ctrl.fDerivativeConstant			:= 0;
Ctrl.fMaxOutputRm 					:= 100;
Ctrl.fMinOutputRm					:= 0;
Ctrl.fCOVIncrement					:= 0;
Ctrl.nDampConstant					:= 0;
Ctrl.fNeutralZone					:= 0;
END_METHOD

END_FUNCTION_BLOCK

// ---- Templates/POUs/Trade/AirConditioning/Aggregates/ERC/Plate/FB_BA_AC_ErcPl_02.TcPOU
{region '#Template'}
	{attribute 'Version' := '6.0.0.0'}
	{attribute 'Tags' := '"LCID": "1031", "Text": "AC, Aggregates, ERC, Plate"'}
	{attribute 'Tags' := '"LCID": "1033", "Text": "AC, Aggregates, ERC, Plate"'}
	{attribute 'Using' := '"Type": "Template", "URI": "Priority"'}		 
	{attribute 'Using' := '"Type": "Template", "URI": "BA2_Param"'}
	{attribute 'Using' := '"Type": "Template", "URI": "EC_ID"'}
	{attribute 'Description' := '"LCID": "1031", "Text": "Aggregat Energie Rückgewinnung Platte mit Bypass"'}
	{attribute 'Description' := '"LCID": "1033", "Text": "Aggregate energy recovery plate with bypass"'}
{endregion}
FUNCTION_BLOCK FB_BA_AC_ErcPl_02 EXTENDS FB_BA_View
VAR_INPUT
	fSpTSuA					: REAL;
	fTSuA					: REAL;
	bSyncTSuACtrl			: BOOL;
	fSyncTSuACtrl			: REAL;			
	bDehumf					: BOOL;
	fTExhA					: REAL;
	fTExtA					: REAL;
	fTWth					: REAL;
END_VAR
VAR_OUTPUT
	fPresentValue			: REAL;				
	eAction					: E_BA_Action;
	bActiveSeqCtrl			: BOOL;	
END_VAR
VAR_IN_OUT
	stTSeqLink				: ST_BA_SeqLink;	//	Sequenz Link Struktur	//	Sequence link structure	
	stAggregate				: ST_BA_Aggregate;		
END_VAR
VAR_INPUT CONSTANT
	TSuACtrl				: FB_BA_AC_ErcTSuACtrl;								 
	TExhACtrl				: FB_BA_PID_Sp;		
	DiffPrssSwi				: FB_BA_SensorBinary;							
	IcePrtcRamp				: FB_BA_RampLimitIncrease;								
	Dmp						: FB_BA_ActuatorAnalog;
	ByDmp					: FB_BA_ActuatorAnalog;					
	PlantLock				: FB_BA_PlantLock;		
	Aggregate				: FB_BA_Aggregate;																											 							
END_VAR
VAR
	bPrioSfty				: BOOL;
	bPrioCrit				: BOOL;		
	PrioSwiVal				: FB_BA_PrioSwi_B04;	
	Inv						: FB_BA_Chrct02;	
END_VAR
VAR // added by the converter: edge detectors and wires of the graphical bodies
    _s1, _s2 : ST_BA_Analog;
    _w1 : ANY;
END_VAR

SUPER^(); // FB_BA_View
Aggregate(stAggregate := stAggregate); // FB_BA_Aggregate
PlantLock(); // FB_BA_PlantLock
bPrioSfty := PlantLock.bPrioHigh OR PlantLock.bPrioLocalHigh;
bPrioCrit := PlantLock.bPrioMedium OR PlantLock.bPrioLocalMedium;
PrioSwiVal(
    bEn01 := Aggregate.arrPriorities[Priority.nLifeSafety],
    bVal01 := Aggregate.bValue,
    bEn02 := Aggregate.arrPriorities[Priority.nCritical],
    bVal02 := Aggregate.bValue,
    bEn03 := Aggregate.arrPriorities[Priority.nProgram],
    bVal03 := Aggregate.bValue); // FB_BA_PrioSwi_B04
TSuACtrl(
    bEn := PrioSwiVal.bVal,
    fSpTSuA := fSpTSuA,
    fTSuA := fTSuA,
    bSync := bSyncTSuACtrl,
    fSync := fSyncTSuACtrl,
    bDehumf := bDehumf,
    fTExtA := fTExtA,
    fTWth := fTWth,
    stSeqLink := stTSeqLink); // FB_BA_AC_ErcTSuACtrl
eAction := TSuACtrl.eAction;
bActiveSeqCtrl := TSuACtrl.bIsActive;
TExhACtrl(bEn := BA2_Param.bDlyStartPLC, fX := fTExhA, bSync := PrioSwiVal.bVal, fSync := 100); // FB_BA_PID_Sp
DiffPrssSwi(); // FB_BA_SensorBinary
IcePrtcRamp(bEn := BA2_Param.bDlyStartPLC, bTrig := DiffPrssSwi.bPresentValue); // FB_BA_RampLimitIncrease
_w1 := MIN(TSuACtrl.fY, TExhACtrl.fY, IcePrtcRamp.fY);
// compose _s1 : ST_BA_Analog
_s1.bEnSfty := Aggregate.arrPriorities[Priority.nLifeSafety];
_s1.fValSfty := _w1;
_s1.bEnCrit := Aggregate.arrPriorities[Priority.nCritical];
_s1.fValCrit := _w1;
_s1.bEnPgm := Aggregate.arrPriorities[Priority.nProgram];
_s1.fValPgm := _w1;
Dmp(stCmd := _s1); // FB_BA_ActuatorAnalog
fPresentValue := Dmp.fMdlt;
Inv(fX := fPresentValue, fX01 := 0, fX02 := 100, fY01 := 100, fY02 := 0, fYMin := 0, fYMax := 100); // FB_BA_Chrct02
// compose _s2 : ST_BA_Analog
_s2.bEnSfty := Aggregate.arrPriorities[Priority.nLifeSafety];
_s2.fValSfty := Inv.fCalcVal;
_s2.bEnCrit := Aggregate.arrPriorities[Priority.nCritical];
_s2.fValCrit := Inv.fCalcVal;
_s2.bEnPgm := Aggregate.arrPriorities[Priority.nProgram];
_s2.fValPgm := Inv.fCalcVal;
ByDmp(stCmd := _s2); // FB_BA_ActuatorAnalog

METHOD FB_init : BOOL
VAR_INPUT
	bInitRetains : BOOL; // if TRUE, the retain variables are initialized (warm start / cold start)
	bInCopyCode : BOOL;  // if TRUE, the instance afterwards gets moved into the copy code (online change)
END_VAR
PlantLock.Parent								:= THIS^;		

TSuACtrl.iParent								:= THIS^;	 
TSuACtrl.iLabel									:= LblCtl_SupplyAirTemperatureControl;   
TSuACtrl.sObjectName							:= '{Idx=21}';						 
TSuACtrl.eDPADMode								:= E_BA_DPADMode.eInclude;								

TExhACtrl.iParent								:= THIS^;	
TExhACtrl.iLabel								:= LblCtl_ExhaustAirTemperatureControl;  
TExhACtrl.sObjectName							:= '{Idx=22}';						 
TExhACtrl.eDPADMode								:= E_BA_DPADMode.eInclude;	
TExhACtrl.Sp.fValueRm 							:= 3.0;
TExhACtrl.Ctrl.eActionRm						:= E_BA_Action.eDirect;			

DiffPrssSwi.iParent								:= THIS^;	
DiffPrssSwi.iLabel								:= LblAgg_PressureDifferential;  
DiffPrssSwi.sObjectName							:= '{Idx=21}';						 
DiffPrssSwi.eDPADMode							:= E_BA_DPADMode.eInclude;
DiffPrssSwi.Input.iLabel						:= LblFun_OperationalMessage;   
DiffPrssSwi.Input.sObjectName					:= '{Idx=01}';						 
DiffPrssSwi.Input.ePolarity						:= E_BA_Polarity.eReverse;
DiffPrssSwi.Input.sActiveText 					:= txtEvent_Triggered;
DiffPrssSwi.Input.sInactiveText 				:= txtEvent_Normal;
DiffPrssSwi.Input.nEventClassID					:= EC_ID.NC30;
DiffPrssSwi.Input.aEventTransitionText[1]		:= txtEvent_Triggered;
DiffPrssSwi.Input.aEventTransitionText[2]		:= txtEvent_Error;
DiffPrssSwi.Input.aEventTransitionText[3]		:= txtEvent_Normal;
DiffPrssSwi.Input.bEventDetectionEnable			:= TRUE;
DiffPrssSwi.Input.eEnPlantLock					:= E_BA_LockPriority.eNoLock;	


IcePrtcRamp.iParent								:= THIS^;	
IcePrtcRamp.iLabel								:= LblCtl_EnergyRecoveryDeicingRamp;   
IcePrtcRamp.sObjectName							:= '{Idx=21}';						 
IcePrtcRamp.eDPADMode							:= E_BA_DPADMode.eInclude;
IcePrtcRamp.TiUp.fValueRm						:= 1200;

Dmp.iParent										:= THIS^;
Dmp.iLabel										:= LblAgg_VentilationDamperSupplyAir;   										 
Dmp.sObjectName									:= '{Idx=21}';						 
Dmp.eDPADMode									:= E_BA_DPADMode.eInclude;
Dmp.Mdlt.fResolution 							:= 0.003814755;
Dmp.Mdlt.fScaleOffset 							:= 0;

ByDmp.iParent									:= THIS^;
ByDmp.iLabel									:= LblAgg_VentilationDamperBypassAir;   									 
ByDmp.sObjectName								:= '{Idx=22}';						 
ByDmp.eDPADMode									:= E_BA_DPADMode.eInclude;
ByDmp.Mdlt.fResolution 							:= 0.003814755;
ByDmp.Mdlt.fScaleOffset 						:= 0;
END_METHOD

END_FUNCTION_BLOCK

// ---- Templates/POUs/Trade/AirConditioning/Aggregates/Fan/FB_BA_AC_FanCtl.TcPOU
{region '#Template'}
	{attribute 'Version' := '6.0.0.0'}
	{attribute 'Tags' := '"LCID": "1031", "Text": "AC, Aggregate, Ventilator"'}
	{attribute 'Tags' := '"LCID": "1033", "Text": "AC, Aggregate, Fan"'}
	{attribute 'Using' := '"Type": "Template", "URI": "Priority"'}		 
	{attribute 'Using' := '"Type": "Template", "URI": "EC_ID"'}
	{attribute 'Using' := '"Type": "Template", "URI": "BA2_Param"'}
	{attribute 'Description' := '"LCID": "1031", "Text": "Ventilator modulierend mit Regler erweitert"'}
	{attribute 'Description' := '"LCID": "1033", "Text": "Fan modulating with controller extended"'}
{endregion}		 
FUNCTION_BLOCK FB_BA_AC_FanCtl EXTENDS FB_BA_MotCtl
VAR_INPUT
	bDamperOpen				: BOOL;
END_VAR
VAR_IN_OUT
	stAggregate				: ST_BA_Aggregate;	
END_VAR
VAR_INPUT CONSTANT
	ThOvrld					: FB_BA_BI_Raw;							
	MntnSwi					: FB_BA_BI_Raw;
	Aggregate				: FB_BA_Aggregate;																											 								
END_VAR
VAR
	PrioSwiDamper			: FB_BA_PrioSwi_UDI04;
END_VAR
VAR // added by the converter: edge detectors and wires of the graphical bodies
    _s1 : ST_BA_Mdlt;
END_VAR

Aggregate(stAggregate := stAggregate); // FB_BA_Aggregate
ThOvrld(); // FB_BA_BI_Raw
MntnSwi(); // FB_BA_BI_Raw
PrioSwiDamper(
    bEn01 := NOT bDamperOpen,
    nVal01 := E_BA_Mdlt.eOff,
    bEn03 := Aggregate.arrPriorities[Priority.nCritical],
    nVal03 := MAX(1,Aggregate.nValue)); // FB_BA_PrioSwi_UDI04
// compose _s1 : ST_BA_Mdlt
_s1.bEnSfty := Aggregate.arrPriorities[Priority.nLifeSafety];
_s1.eValSfty := MAX(1,Aggregate.nValue);
_s1.bEnCrit := PrioSwiDamper.bQ;
_s1.eValCrit := PrioSwiDamper.nVal;
_s1.bEnPgm := Aggregate.arrPriorities[Priority.nProgram];
_s1.eValPgm := MAX(1,Aggregate.nValue);
SUPER^(stCmd := _s1); // FB_BA_MotCtl

METHOD FB_init : BOOL
VAR_INPUT
	bInitRetains : BOOL; // if TRUE, the retain variables are initialized (warm start / cold start)
	bInCopyCode : BOOL;  // if TRUE, the instance afterwards gets moved into the copy code (online change)
END_VAR
ThOvrld.iParent						:= THIS^;
ThOvrld.iLabel						:= LblFun_Fault;  
ThOvrld.ePolarity					:= E_BA_Polarity.eReverse;
ThOvrld.sActiveText 				:= txtEvent_Triggered;
ThOvrld.sInactiveText 				:= txtEvent_Normal;
ThOvrld.nEventClassID				:= EC_ID.NC30;
ThOvrld.stTimeDelay.nToNormal		:= BA2_Param.nDefTimeDelay_ToNormal;
ThOvrld.stTimeDelay.nToAbnormal		:= BA2_Param.nDefTimeDelay_ToAbnormal;
ThOvrld.bAlarmValue					:= TRUE;
ThOvrld.aEventTransitionText[1]		:= txtEvent_Triggered;
ThOvrld.aEventTransitionText[2]		:= txtEvent_Error;
ThOvrld.aEventTransitionText[3]		:= txtEvent_Normal;
ThOvrld.bEventDetectionEnable		:= TRUE;
ThOvrld.eEnPlantLock				:= E_BA_LockPriority.eLocalMedium;	

MntnSwi.iParent						:= THIS^;
MntnSwi.iLabel						:= LblFun_MaintenanceMessage;  
MntnSwi.ePolarity					:= E_BA_Polarity.eReverse;
MntnSwi.sActiveText 				:= txtEvent_Maintenace;
MntnSwi.sInactiveText 				:= txtEvent_Normal;
MntnSwi.nEventClassID				:= EC_ID.NC50;
MntnSwi.stTimeDelay.nToNormal		:= BA2_Param.nDefTimeDelay_ToNormal;
MntnSwi.stTimeDelay.nToAbnormal		:= BA2_Param.nDefTimeDelay_ToAbnormal;
MntnSwi.bAlarmValue					:= TRUE;
MntnSwi.aEventTransitionText[1]		:= txtEvent_Disturb;
MntnSwi.aEventTransitionText[2]		:= txtEvent_None;
MntnSwi.aEventTransitionText[3]		:= txtEvent_Normal;
MntnSwi.bEventDetectionEnable		:= TRUE;
MntnSwi.eEnPlantLock				:= E_BA_LockPriority.eLocalMedium;
END_METHOD

END_FUNCTION_BLOCK

// ---- Templates/POUs/Universal/Motor/Control/FB_BA_MotCtl.TcPOU
{region '#Template'}
	{attribute 'Version' := '5.0.0.0'}
	{attribute 'Tags' := '"LCID": "1031", "Text": "Universal, Motor, Aggregate"'}
	{attribute 'Tags' := '"LCID": "1033", "Text": "Universal, Motor, Aggregate"'}
	{attribute 'Using' := '"Type": "Template", "URI": "EC_ID"'}
	{attribute 'Using' := '"Type": "Template", "URI": "BA2_Param"'}
	{attribute 'Description' := '"LCID": "1031", "Text": "Motor modulierend mit Regler"'}
	{attribute 'Description' := '"LCID": "1033", "Text": "Motor modulating with controller"'}
{endregion}		
FUNCTION_BLOCK FB_BA_MotCtl EXTENDS FB_BA_View
VAR_INPUT
	fIn				: REAL;	// Istwert Regler // Actual value controller	
	stCmd			: ST_BA_Mdlt;
END_VAR
VAR_OUTPUT
	bCmd			: BOOL;
	fMdlt			: REAL;
	bDst			: BOOL;
	eActivePrio		: E_BA_Priority;
END_VAR

VAR_INPUT CONSTANT
	Dst				: FB_BA_BI_Raw;
	Cmd				: FB_BA_BO_Raw;								 
	Mdlt			: FB_BA_AO_Raw;							
	Sp				: FB_BA_AV_Op;		 
	Ctrl			: FB_BA_Loop;		
	PlantLock		: FB_BA_PlantLock;														
END_VAR
VAR
	bPrioSfty					: BOOL;
	bPrioCrit					: BOOL;	
	
	PrioSwiVal					: FB_BA_PrioSwi_UDI04;	

	MuxCmd						: FB_BA_MMUX_B04;
	MuxMdlt						: FB_BA_MMUX_R04;
	fMax						: REAL;
	fMin						: REAL;		
END_VAR
VAR // added by the converter: edge detectors and wires of the graphical bodies
    _w1, _w2 : ANY;
END_VAR

